LIN {X 0,Y 406.447,Z 396.018,A -85,B 0,C 180,E1 17983.42,E2 17983.42} C_VEL
LIN {X 0,Y 407.106,Z 396.844,A -85,B 0,C 180,E1 17981.451,E2 17981.451} C_VEL
LIN {X 0,Y 409.582,Z 400.807,A -85,B 0,C 180,E1 17978.37,E2 17978.37} C_VEL
LIN {X 0,Y 412.361,Z 402.697,A -85,B 0,C 180,E1 17976.455,E2 17976.455} C_VEL
LIN {X 0,Y 414.579,Z 406.468,A -85,B 0,C 180,E1 17975.036,E2 17975.036} C_VEL
LIN {X 0,Y 417.386,Z 409.126,A -85,B 0,C 180,E1 17973.649,E2 17973.649} C_VEL
LIN {X 0,Y 421.803,Z 415.235,A -85,B 0,C 180,E1 17971.701,E2 17971.701} C_VEL
LIN {X 0,Y 425.14,Z 419.754,A -85,B 0,C 180,E1 17970.443,E2 17970.443} C_VEL
LIN {X 0,Y 429.609,Z 426.182,A -85,B 0,C 180,E1 17968.891,E2 17968.891} C_VEL
LIN {X 0,Y 436.176,Z 435.925,A -85,B 0,C 180,E1 17966.897,E2 17966.897} C_VEL
LIN {X 0,Y 443.079,Z 446.923,A -85,B 0,C 180,E1 17965.028,E2 17965.028} C_VEL
LIN {X 0,Y 450.903,Z 460.1,A -85,B 0,C 180,E1 17963.124,E2 17963.124} C_VEL
LIN {X 0,Y 451.957,Z 462.413,A -85,B 0,C 180,E1 17962.867,E2 17962.867} C_VEL
LIN {X 0,Y 443.085,Z 650.195,A -85,B 0,C 180,E1 17959.257,E2 17959.257} C_VEL
LIN {X 0,Y 439.216,Z 737.669,A -85,B 0,C 180,E1 17957.582,E2 17957.582} C_VEL
LIN {X 0,Y 437.021,Z 761.221,A -85,B 0,C 180,E1 17956.942,E2 17956.942} C_VEL
LIN {X 0,Y 434.323,Z 783.972,A -85,B 0,C 180,E1 17956.104,E2 17956.104} C_VEL
LIN {X 0,Y 431.268,Z 805.02,A -85,B 0,C 180,E1 17955.098,E2 17955.098} C_VEL
LIN {X 0,Y 427.411,Z 828.313,A -85,B 0,C 180,E1 17953.71,E2 17953.71} C_VEL
LIN {X 0,Y 423.869,Z 847.343,A -85,B 0,C 180,E1 17952.338,E2 17952.338} C_VEL
LIN {X 0,Y 419.579,Z 868.496,A -85,B 0,C 180,E1 17950.521,E2 17950.521} C_VEL
LIN {X 0,Y 415.449,Z 887.81,A -85,B 0,C 180,E1 17948.563,E2 17948.563} C_VEL
LIN {X 0,Y 411.376,Z 906.017,A -85,B 0,C 180,E1 17946.377,E2 17946.377} C_VEL
LIN {X 0,Y 407.459,Z 923.411,A -85,B 0,C 180,E1 17943.962,E2 17943.962} C_VEL
LIN {X 0,Y 404.032,Z 938.688,A -85,B 0,C 180,E1 17941.481,E2 17941.481} C_VEL
LIN {X 0,Y 400.669,Z 954.261,A -85,B 0,C 180,E1 17938.55,E2 17938.55} C_VEL
LIN {X 0,Y 398.109,Z 966.963,A -85,B 0,C 180,E1 17935.756,E2 17935.756} C_VEL
LIN {X 0,Y 395.862,Z 979.241,A -85,B 0,C 180,E1 17932.58,E2 17932.58} C_VEL
LIN {X 0,Y 394.305,Z 989.174,A -85,B 0,C 180,E1 17929.559,E2 17929.559} C_VEL
LIN {X 0,Y 393.186,Z 997.73,A -85,B 0,C 180,E1 17926.399,E2 17926.399} C_VEL
LIN {X 0,Y 392.494,Z 1004.736,A -85,B 0,C 180,E1 17923.258,E2 17923.258} C_VEL
LIN {X 0,Y 392.088,Z 1010.3,A -85,B 0,C 180,E1 17919.989,E2 17919.989} C_VEL
LIN {X 0,Y 391.941,Z 1013.854,A -85,B 0,C 180,E1 17917.184,E2 17917.184} C_VEL
LIN {X 0,Y 391.914,Z 1016.518,A -85,B 0,C 180,E1 17913.954,E2 17913.954} C_VEL
LIN {X 0,Y 391.905,Z 1017.533,A -85,B 0,C 180,E1 17911.173,E2 17911.173} C_VEL
LIN {X 0,Y 391.911,Z 1017.466,A -85,B 0,C 180,E1 17908.396,E2 17908.396} C_VEL
LIN {X 0,Y 391.917,Z 1015.846,A -85,B 0,C 180,E1 17905.028,E2 17905.028} C_VEL
LIN {X 0,Y 391.978,Z 1013.228,A -85,B 0,C 180,E1 17902.234,E2 17902.234} C_VEL
LIN {X 0,Y 392.194,Z 1008.814,A -85,B 0,C 180,E1 17898.981,E2 17898.981} C_VEL
LIN {X 0,Y 392.64,Z 1002.949,A -85,B 0,C 180,E1 17895.854,E2 17895.854} C_VEL
LIN {X 0,Y 393.449,Z 995.665,A -85,B 0,C 180,E1 17892.707,E2 17892.707} C_VEL
LIN {X 0,Y 394.712,Z 986.541,A -85,B 0,C 180,E1 17889.544,E2 17889.544} C_VEL
LIN {X 0,Y 396.55,Z 975.718,A -85,B 0,C 180,E1 17886.37,E2 17886.37} C_VEL
LIN {X 0,Y 398.776,Z 964.082,A -85,B 0,C 180,E1 17883.498,E2 17883.498} C_VEL
LIN {X 0,Y 401.77,Z 949.865,A -85,B 0,C 180,E1 17880.484,E2 17880.484} C_VEL
LIN {X 0,Y 404.955,Z 935.505,A -85,B 0,C 180,E1 17877.874,E2 17877.874} C_VEL
LIN {X 0,Y 408.783,Z 918.746,A -85,B 0,C 180,E1 17875.262,E2 17875.262} C_VEL
LIN {X 0,Y 412.641,Z 901.934,A -85,B 0,C 180,E1 17872.999,E2 17872.999} C_VEL
LIN {X 0,Y 416.749,Z 883.443,A -85,B 0,C 180,E1 17870.883,E2 17870.883} C_VEL
LIN {X 0,Y 420.829,Z 864.613,A -85,B 0,C 180,E1 17869.03,E2 17869.03} C_VEL
LIN {X 0,Y 424.656,Z 845.158,A -85,B 0,C 180,E1 17867.422,E2 17867.422} C_VEL
LIN {X 0,Y 428.329,Z 825.276,A -85,B 0,C 180,E1 17866.023,E2 17866.023} C_VEL
LIN {X 0,Y 431.758,Z 803.746,A -85,B 0,C 180,E1 17864.789,E2 17864.789} C_VEL
LIN {X 0,Y 434.972,Z 780.771,A -85,B 0,C 180,E1 17863.734,E2 17863.734} C_VEL
LIN {X 0,Y 437.348,Z 759.57,A -85,B 0,C 180,E1 17862.988,E2 17862.988} C_VEL
LIN {X 0,Y 439.399,Z 734.535,A -85,B 0,C 180,E1 17862.352,E2 17862.352} C_VEL
LIN {X 0,Y 448.069,Z 525.057,A -85,B 0,C 180,E1 17858.43,E2 17858.43} C_VEL
LIN {X 0,Y 450.713,Z 461.917,A -85,B 0,C 180,E1 17857.213,E2 17857.213} C_VEL
LIN {X 0,Y 440.051,Z 445.277,A -85,B 0,C 180,E1 17854.969,E2 17854.969} C_VEL
LIN {X 0,Y 429.028,Z 429.211,A -85,B 0,C 180,E1 17852.452,E2 17852.452} C_VEL
LIN {X 0,Y 421.006,Z 418.219,A -85,B 0,C 180,E1 17850.467,E2 17850.467} C_VEL
LIN {X 0,Y 413.797,Z 408.572,A -85,B 0,C 180,E1 17848.543,E2 17848.543} C_VEL
LIN {X 0,Y 410.464,Z 404.237,A -85,B 0,C 180,E1 17847.608,E2 17847.608} C_VEL
LIN {X 0,Y 406.022,Z 398.588,A -85,B 0,C 180,E1 17846.312,E2 17846.312} C_VEL
LIN {X 0,Y 401.849,Z 393.423,A -85,B 0,C 180,E1 17845.023,E2 17845.023} C_VEL
LIN {X 0,Y 398.003,Z 388.428,A -85,B 0,C 180,E1 17843.778,E2 17843.778} C_VEL
LIN {X 0,Y 394.851,Z 385.59,A -85,B 0,C 180,E1 17842.755,E2 17842.755} C_VEL
LIN {X 0,Y 393.726,Z 383.145,A -85,B 0,C 180,E1 17842.233,E2 17842.233} C_VEL
LIN {X 0,Y 393.56,Z 382.126,A -85,B 0,C 180,E1 17841.772,E2 17841.772} C_VEL
LIN {X 0,Y 393.536,Z 382.017,A -85,B 0,C 180,E1 17837.7,E2 17837.7} C_VEL
LIN {X 0,Y 393.524,Z 382.017,A -85,B 0,C 180,E1 17833.817,E2 17833.817} C_VEL
LIN {X 0,Y 393.51,Z 382.027,A -85,B 0,C 180,E1 17829.949,E2 17829.949} C_VEL
LIN {X 0,Y 393.504,Z 382.032,A -85,B 0,C 180,E1 17826.126,E2 17826.126} C_VEL
LIN {X 0,Y 393.503,Z 382.025,A -85,B 0,C 180,E1 17822.184,E2 17822.184} C_VEL
LIN {X 0,Y 393.507,Z 382.019,A -85,B 0,C 180,E1 17818.252,E2 17818.252} C_VEL
LIN {X 0,Y 393.516,Z 382.015,A -85,B 0,C 180,E1 17814.313,E2 17814.313} C_VEL
LIN {X 0,Y 393.537,Z 382.014,A -85,B 0,C 180,E1 17810.494,E2 17810.494} C_VEL
LIN {X 0,Y 393.558,Z 382.012,A -85,B 0,C 180,E1 17806.632,E2 17806.632} C_VEL
LIN {X 0,Y 393.558,Z 382.015,A -85,B 0,C 180,E1 17802.707,E2 17802.707} C_VEL
LIN {X 0,Y 393.559,Z 382.02,A -85,B 0,C 180,E1 17798.697,E2 17798.697} C_VEL
LIN {X 0,Y 393.552,Z 382.026,A -85,B 0,C 180,E1 17794.734,E2 17794.734} C_VEL
LIN {X 0,Y 393.542,Z 382.027,A -85,B 0,C 180,E1 17790.803,E2 17790.803} C_VEL
LIN {X 0,Y 393.535,Z 382.021,A -85,B 0,C 180,E1 17786.889,E2 17786.889} C_VEL
LIN {X 0,Y 393.531,Z 382.016,A -85,B 0,C 180,E1 17782.911,E2 17782.911} C_VEL
LIN {X 0,Y 393.535,Z 382.014,A -85,B 0,C 180,E1 17778.981,E2 17778.981} C_VEL
LIN {X 0,Y 393.539,Z 382.025,A -85,B 0,C 180,E1 17774.928,E2 17774.928} C_VEL
LIN {X 0,Y 393.544,Z 382.021,A -85,B 0,C 180,E1 17770.95,E2 17770.95} C_VEL
LIN {X 0,Y 393.55,Z 382.014,A -85,B 0,C 180,E1 17767.016,E2 17767.016} C_VEL
LIN {X 0,Y 393.585,Z 382.191,A -85,B 0,C 180,E1 17765.366,E2 17765.366} C_VEL
LIN {X 0,Y 393.904,Z 383.571,A -85,B 0,C 180,E1 17764.927,E2 17764.927} C_VEL
LIN {X 0,Y 395.652,Z 386.503,A -85,B 0,C 180,E1 17764.272,E2 17764.272} C_VEL
LIN {X 0,Y 398.818,Z 388.946,A -85,B 0,C 180,E1 17763.281,E2 17763.281} C_VEL
LIN {X 0,Y 401.093,Z 392.587,A -85,B 0,C 180,E1 17762.52,E2 17762.52} C_VEL
LIN {X 0,Y 404.021,Z 395.14,A -85,B 0,C 180,E1 17761.639,E2 17761.639} C_VEL
LIN {X 0,Y 406.774,Z 399.093,A -85,B 0,C 180,E1 17760.786,E2 17760.786} C_VEL
LIN {X 0,Y 409.03,Z 401.334,A -85,B 0,C 180,E1 17760.148,E2 17760.148} C_VEL
LIN {X 0,Y 412.363,Z 405.67,A -85,B 0,C 180,E1 17759.203,E2 17759.203} C_VEL
LIN {X 0,Y 414.226,Z 407.789,A -85,B 0,C 180,E1 17758.703,E2 17758.703} C_VEL
LIN {X 0,Y 419.171,Z 413.919,A -85,B 0,C 180,E1 17757.406,E2 17757.406} C_VEL
LIN {X 0,Y 423.928,Z 420.03,A -85,B 0,C 180,E1 17756.204,E2 17756.204} C_VEL
LIN {X 0,Y 431.744,Z 430.135,A -85,B 0,C 180,E1 17754.34,E2 17754.34} C_VEL
LIN {X 0,Y 442.645,Z 445.003,A -85,B 0,C 180,E1 17751.946,E2 17751.946} C_VEL
LIN {X 0,Y 450.53,Z 456.58,A -85,B 0,C 180,E1 17750.328,E2 17750.328} C_VEL
LIN {X 0,Y 442.652,Z 641.056,A -85,B 0,C 180,E1 17746.873,E2 17746.873} C_VEL
LIN {X 0,Y 441.678,Z 648.751,A -85,B 0,C 180,E1 17746.826,E2 17746.826} C_VEL
LIN {X 0,Y 436.634,Z 669.324,A -85,B 0,C 180,E1 17747.051,E2 17747.051} C_VEL
LIN {X 0,Y 435.857,Z 675.927,A -85,B 0,C 180,E1 17747,E2 17747} C_VEL
LIN {X 0,Y 433.839,Z 717.756,A -85,B 0,C 180,E1 17746.18,E2 17746.18} C_VEL
LIN {X 0,Y 431.82,Z 739.993,A -85,B 0,C 180,E1 17745.546,E2 17745.546} C_VEL
LIN {X 0,Y 429.069,Z 763.419,A -85,B 0,C 180,E1 17744.641,E2 17744.641} C_VEL
LIN {X 0,Y 426.277,Z 782.547,A -85,B 0,C 180,E1 17743.7,E2 17743.7} C_VEL
LIN {X 0,Y 422.53,Z 804.668,A -85,B 0,C 180,E1 17742.362,E2 17742.362} C_VEL
LIN {X 0,Y 418.935,Z 823.202,A -85,B 0,C 180,E1 17741.003,E2 17741.003} C_VEL
LIN {X 0,Y 414.415,Z 844.319,A -85,B 0,C 180,E1 17739.159,E2 17739.159} C_VEL
LIN {X 0,Y 410.247,Z 862.498,A -85,B 0,C 180,E1 17737.274,E2 17737.274} C_VEL
LIN {X 0,Y 405.893,Z 880.407,A -85,B 0,C 180,E1 17735.084,E2 17735.084} C_VEL
LIN {X 0,Y 401.728,Z 897.125,A -85,B 0,C 180,E1 17732.707,E2 17732.707} C_VEL
LIN {X 0,Y 397.837,Z 912.385,A -85,B 0,C 180,E1 17730.14,E2 17730.14} C_VEL
LIN {X 0,Y 394.34,Z 926.605,A -85,B 0,C 180,E1 17727.38,E2 17727.38} C_VEL
LIN {X 0,Y 391.42,Z 938.864,A -85,B 0,C 180,E1 17724.573,E2 17724.573} C_VEL
LIN {X 0,Y 388.851,Z 950.67,A -85,B 0,C 180,E1 17721.42,E2 17721.42} C_VEL
LIN {X 0,Y 386.984,Z 960.23,A -85,B 0,C 180,E1 17718.37,E2 17718.37} C_VEL
LIN {X 0,Y 385.494,Z 969.457,A -85,B 0,C 180,E1 17714.81,E2 17714.81} C_VEL
LIN {X 0,Y 384.655,Z 976.186,A -85,B 0,C 180,E1 17711.582,E2 17711.582} C_VEL
LIN {X 0,Y 384.17,Z 981.649,A -85,B 0,C 180,E1 17708.147,E2 17708.147} C_VEL
LIN {X 0,Y 383.977,Z 985.556,A -85,B 0,C 180,E1 17704.716,E2 17704.716} C_VEL
LIN {X 0,Y 383.93,Z 987.8,A -85,B 0,C 180,E1 17701.36,E2 17701.36} C_VEL
LIN {X 0,Y 383.915,Z 988.609,A -85,B 0,C 180,E1 17698.08,E2 17698.08} C_VEL
LIN {X 0,Y 383.926,Z 987.87,A -85,B 0,C 180,E1 17694.676,E2 17694.676} C_VEL
LIN {X 0,Y 383.978,Z 985.703,A -85,B 0,C 180,E1 17691.318,E2 17691.318} C_VEL
LIN {X 0,Y 384.167,Z 981.866,A -85,B 0,C 180,E1 17687.882,E2 17687.882} C_VEL
LIN {X 0,Y 384.636,Z 976.512,A -85,B 0,C 180,E1 17684.451,E2 17684.451} C_VEL
LIN {X 0,Y 385.471,Z 969.833,A -85,B 0,C 180,E1 17681.212,E2 17681.212} C_VEL
LIN {X 0,Y 386.915,Z 960.986,A -85,B 0,C 180,E1 17677.74,E2 17677.74} C_VEL
LIN {X 0,Y 388.714,Z 951.69,A -85,B 0,C 180,E1 17674.735,E2 17674.735} C_VEL
LIN {X 0,Y 391.407,Z 939.423,A -85,B 0,C 180,E1 17671.408,E2 17671.408} C_VEL
LIN {X 0,Y 394.527,Z 926.457,A -85,B 0,C 180,E1 17668.425,E2 17668.425} C_VEL
LIN {X 0,Y 398.171,Z 911.785,A -85,B 0,C 180,E1 17665.59,E2 17665.59} C_VEL
LIN {X 0,Y 402.352,Z 895.45,A -85,B 0,C 180,E1 17662.886,E2 17662.886} C_VEL
LIN {X 0,Y 406.463,Z 879.226,A -85,B 0,C 180,E1 17660.596,E2 17660.596} C_VEL
LIN {X 0,Y 410.926,Z 860.86,A -85,B 0,C 180,E1 17658.383,E2 17658.383} C_VEL
LIN {X 0,Y 415.401,Z 841.777,A -85,B 0,C 180,E1 17656.429,E2 17656.429} C_VEL
LIN {X 0,Y 419.495,Z 822.459,A -85,B 0,C 180,E1 17654.776,E2 17654.776} C_VEL
LIN {X 0,Y 423.374,Z 802.677,A -85,B 0,C 180,E1 17653.339,E2 17653.339} C_VEL
LIN {X 0,Y 426.861,Z 781.831,A -85,B 0,C 180,E1 17652.102,E2 17652.102} C_VEL
LIN {X 0,Y 430.013,Z 760.158,A -85,B 0,C 180,E1 17651.053,E2 17651.053} C_VEL
LIN {X 0,Y 432.527,Z 738.038,A -85,B 0,C 180,E1 17650.233,E2 17650.233} C_VEL
LIN {X 0,Y 434.647,Z 712.891,A -85,B 0,C 180,E1 17649.563,E2 17649.563} C_VEL
LIN {X 0,Y 444.951,Z 502.944,A -85,B 0,C 180,E1 17645.5,E2 17645.5} C_VEL
LIN {X 0,Y 447.109,Z 460.805,A -85,B 0,C 180,E1 17644.65,E2 17644.65} C_VEL
LIN {X 0,Y 439.45,Z 449.084,A -85,B 0,C 180,E1 17642.739,E2 17642.739} C_VEL
LIN {X 0,Y 432.726,Z 439.435,A -85,B 0,C 180,E1 17640.861,E2 17640.861} C_VEL
LIN {X 0,Y 426.889,Z 431.418,A -85,B 0,C 180,E1 17639.027,E2 17639.027} C_VEL
LIN {X 0,Y 423.277,Z 426.612,A -85,B 0,C 180,E1 17637.75,E2 17637.75} C_VEL
LIN {X 0,Y 419.427,Z 421.563,A -85,B 0,C 180,E1 17636.242,E2 17636.242} C_VEL
LIN {X 0,Y 416.196,Z 417.577,A -85,B 0,C 180,E1 17634.797,E2 17634.797} C_VEL
LIN {X 0,Y 415.277,Z 416.109,A -85,B 0,C 180,E1 17634.335,E2 17634.335} C_VEL
LIN {X 0,Y 412.079,Z 412.864,A -85,B 0,C 180,E1 17632.612,E2 17632.612} C_VEL
LIN {X 0,Y 410.451,Z 410.075,A -85,B 0,C 180,E1 17631.511,E2 17631.511} C_VEL
LIN {X 0,Y 406.913,Z 407.011,A -85,B 0,C 180,E1 17628.52,E2 17628.52} C_VEL
LIN {X 0,Y 405.709,Z 404.273,A -85,B 0,C 180,E1 17626.315,E2 17626.315} C_VEL
LIN {X 0,Y 405.34,Z 403.948,A -85,B 0,C 180,E1 17623.374,E2 17623.374} C_VEL
LIN {X 0,Y 405.911,Z 404.661,A -85,B 0,C 180,E1 17621.622,E2 17621.622} C_VEL
LIN {X 0,Y 408.352,Z 408.698,A -85,B 0,C 180,E1 17618.453,E2 17618.453} C_VEL
LIN {X 0,Y 410.84,Z 410.578,A -85,B 0,C 180,E1 17616.667,E2 17616.667} C_VEL
LIN {X 0,Y 413.282,Z 414.449,A -85,B 0,C 180,E1 17615.105,E2 17615.105} C_VEL
LIN {X 0,Y 415.69,Z 416.816,A -85,B 0,C 180,E1 17613.886,E2 17613.886} C_VEL
LIN {X 0,Y 419.948,Z 422.878,A -85,B 0,C 180,E1 17611.951,E2 17611.951} C_VEL
LIN {X 0,Y 422.937,Z 427.073,A -85,B 0,C 180,E1 17610.779,E2 17610.779} C_VEL
LIN {X 0,Y 428.371,Z 434.95,A -85,B 0,C 180,E1 17608.869,E2 17608.869} C_VEL
LIN {X 0,Y 435.097,Z 445.542,A -85,B 0,C 180,E1 17606.805,E2 17606.805} C_VEL
LIN {X 0,Y 441.885,Z 456.681,A -85,B 0,C 180,E1 17604.96,E2 17604.96} C_VEL
LIN {X 0,Y 447.17,Z 466.131,A -85,B 0,C 180,E1 17603.635,E2 17603.635} C_VEL
LIN {X 0,Y 437.799,Z 653.274,A -85,B 0,C 180,E1 17600,E2 17600} C_VEL
LIN {X 0,Y 433.839,Z 737.361,A -85,B 0,C 180,E1 17598.368,E2 17598.368} C_VEL
LIN {X 0,Y 431.556,Z 760.907,A -85,B 0,C 180,E1 17597.724,E2 17597.724} C_VEL
LIN {X 0,Y 428.741,Z 783.618,A -85,B 0,C 180,E1 17596.884,E2 17596.884} C_VEL
LIN {X 0,Y 425.543,Z 804.601,A -85,B 0,C 180,E1 17595.876,E2 17595.876} C_VEL
LIN {X 0,Y 421.46,Z 828.087,A -85,B 0,C 180,E1 17594.468,E2 17594.468} C_VEL
LIN {X 0,Y 417.618,Z 847.811,A -85,B 0,C 180,E1 17593.03,E2 17593.03} C_VEL
LIN {X 0,Y 413.324,Z 867.93,A -85,B 0,C 180,E1 17591.278,E2 17591.278} C_VEL
LIN {X 0,Y 409.099,Z 886.671,A -85,B 0,C 180,E1 17589.366,E2 17589.366} C_VEL
LIN {X 0,Y 404.842,Z 904.725,A -85,B 0,C 180,E1 17587.19,E2 17587.19} C_VEL
LIN {X 0,Y 400.727,Z 922.148,A -85,B 0,C 180,E1 17584.763,E2 17584.763} C_VEL
LIN {X 0,Y 396.867,Z 938.245,A -85,B 0,C 180,E1 17582.116,E2 17582.116} C_VEL
LIN {X 0,Y 393.38,Z 953.475,A -85,B 0,C 180,E1 17579.213,E2 17579.213} C_VEL
LIN {X 0,Y 390.649,Z 966.145,A -85,B 0,C 180,E1 17576.388,E2 17576.388} C_VEL
LIN {X 0,Y 388.161,Z 978.857,A -85,B 0,C 180,E1 17573.053,E2 17573.053} C_VEL
LIN {X 0,Y 386.486,Z 988.803,A -85,B 0,C 180,E1 17569.971,E2 17569.971} C_VEL
LIN {X 0,Y 385.282,Z 997.376,A -85,B 0,C 180,E1 17566.745,E2 17566.745} C_VEL
LIN {X 0,Y 384.563,Z 1004.083,A -85,B 0,C 180,E1 17563.689,E2 17563.689} C_VEL
LIN {X 0,Y 384.114,Z 1009.854,A -85,B 0,C 180,E1 17560.284,E2 17560.284} C_VEL
LIN {X 0,Y 383.956,Z 1013.372,A -85,B 0,C 180,E1 17557.485,E2 17557.485} C_VEL
LIN {X 0,Y 383.917,Z 1016.07,A -85,B 0,C 180,E1 17554.335,E2 17554.335} C_VEL
LIN {X 0,Y 383.916,Z 1017.207,A -85,B 0,C 180,E1 17551.347,E2 17551.347} C_VEL
LIN {X 0,Y 383.917,Z 1017.19,A -85,B 0,C 180,E1 17548.512,E2 17548.512} C_VEL
LIN {X 0,Y 383.917,Z 1015.781,A -85,B 0,C 180,E1 17545.224,E2 17545.224} C_VEL
LIN {X 0,Y 383.979,Z 1013.093,A -85,B 0,C 180,E1 17542.222,E2 17542.222} C_VEL
LIN {X 0,Y 384.187,Z 1008.986,A -85,B 0,C 180,E1 17539.052,E2 17539.052} C_VEL
LIN {X 0,Y 384.645,Z 1003.203,A -85,B 0,C 180,E1 17535.831,E2 17535.831} C_VEL
LIN {X 0,Y 385.421,Z 996.454,A -85,B 0,C 180,E1 17532.803,E2 17532.803} C_VEL
LIN {X 0,Y 386.78,Z 987.158,A -85,B 0,C 180,E1 17529.421,E2 17529.421} C_VEL
LIN {X 0,Y 388.585,Z 977.068,A -85,B 0,C 180,E1 17526.339,E2 17526.339} C_VEL
LIN {X 0,Y 391.007,Z 965.039,A -85,B 0,C 180,E1 17523.258,E2 17523.258} C_VEL
LIN {X 0,Y 393.96,Z 951.86,A -85,B 0,C 180,E1 17520.342,E2 17520.342} C_VEL
LIN {X 0,Y 397.35,Z 937.204,A -85,B 0,C 180,E1 17517.596,E2 17517.596} C_VEL
LIN {X 0,Y 401.426,Z 920.406,A -85,B 0,C 180,E1 17514.881,E2 17514.881} C_VEL
LIN {X 0,Y 405.309,Z 904.242,A -85,B 0,C 180,E1 17512.644,E2 17512.644} C_VEL
LIN {X 0,Y 409.892,Z 884.772,A -85,B 0,C 180,E1 17510.343,E2 17510.343} C_VEL
LIN {X 0,Y 414.085,Z 866.277,A -85,B 0,C 180,E1 17508.483,E2 17508.483} C_VEL
LIN {X 0,Y 418.252,Z 846.309,A -85,B 0,C 180,E1 17506.789,E2 17506.789} C_VEL
LIN {X 0,Y 422.24,Z 825.708,A -85,B 0,C 180,E1 17505.315,E2 17505.315} C_VEL
LIN {X 0,Y 425.93,Z 803.593,A -85,B 0,C 180,E1 17504.037,E2 17504.037} C_VEL
LIN {X 0,Y 429.289,Z 780.498,A -85,B 0,C 180,E1 17502.972,E2 17502.972} C_VEL
LIN {X 0,Y 431.714,Z 759.649,A -85,B 0,C 180,E1 17502.236,E2 17502.236} C_VEL
LIN {X 0,Y 433.861,Z 734.539,A -85,B 0,C 180,E1 17501.59,E2 17501.59} C_VEL
LIN {X 0,Y 442.99,Z 525.076,A -85,B 0,C 180,E1 17497.63,E2 17497.63} C_VEL
LIN {X 0,Y 445.609,Z 465.785,A -85,B 0,C 180,E1 17496.484,E2 17496.484} C_VEL
LIN {X 0,Y 434.795,Z 448.963,A -85,B 0,C 180,E1 17494.132,E2 17494.132} C_VEL
LIN {X 0,Y 424.828,Z 434.413,A -85,B 0,C 180,E1 17491.776,E2 17491.776} C_VEL
LIN {X 0,Y 415.337,Z 421.227,A -85,B 0,C 180,E1 17489.333,E2 17489.333} C_VEL
LIN {X 0,Y 407.646,Z 411.108,A -85,B 0,C 180,E1 17487.182,E2 17487.182} C_VEL
LIN {X 0,Y 403.271,Z 405.482,A -85,B 0,C 180,E1 17485.872,E2 17485.872} C_VEL
LIN {X 0,Y 399.227,Z 400.458,A -85,B 0,C 180,E1 17484.605,E2 17484.605} C_VEL
LIN {X 0,Y 395.116,Z 395.318,A -85,B 0,C 180,E1 17483.251,E2 17483.251} C_VEL
LIN {X 0,Y 392.162,Z 392.283,A -85,B 0,C 180,E1 17482.247,E2 17482.247} C_VEL
LIN {X 0,Y 390.555,Z 389.517,A -85,B 0,C 180,E1 17481.632,E2 17481.632} C_VEL
LIN {X 0,Y 387.32,Z 387.115,A -85,B 0,C 180,E1 17480.513,E2 17480.513} C_VEL
LIN {X 0,Y 385.698,Z 383.627,A -85,B 0,C 180,E1 17479.694,E2 17479.694} C_VEL
LIN {X 0,Y 385.566,Z 383.038,A -85,B 0,C 180,E1 17479.071,E2 17479.071} C_VEL
LIN {X 0,Y 385.577,Z 383.013,A -85,B 0,C 180,E1 17475.183,E2 17475.183} C_VEL
LIN {X 0,Y 385.59,Z 383.004,A -85,B 0,C 180,E1 17471.214,E2 17471.214} C_VEL
LIN {X 0,Y 385.602,Z 383.005,A -85,B 0,C 180,E1 17467.149,E2 17467.149} C_VEL
LIN {X 0,Y 385.604,Z 383.015,A -85,B 0,C 180,E1 17463.121,E2 17463.121} C_VEL
LIN {X 0,Y 385.619,Z 383.012,A -85,B 0,C 180,E1 17459.108,E2 17459.108} C_VEL
LIN {X 0,Y 385.613,Z 383.003,A -85,B 0,C 180,E1 17454.942,E2 17454.942} C_VEL
LIN {X 0,Y 385.616,Z 383,A -85,B 0,C 180,E1 17450.899,E2 17450.899} C_VEL
LIN {X 0,Y 385.619,Z 383,A -85,B 0,C 180,E1 17446.81,E2 17446.81} C_VEL
LIN {X 0,Y 385.615,Z 383.002,A -85,B 0,C 180,E1 17442.807,E2 17442.807} C_VEL
LIN {X 0,Y 385.619,Z 383.008,A -85,B 0,C 180,E1 17438.715,E2 17438.715} C_VEL
LIN {X 0,Y 385.616,Z 383.016,A -85,B 0,C 180,E1 17434.67,E2 17434.67} C_VEL
LIN {X 0,Y 385.618,Z 383.01,A -85,B 0,C 180,E1 17430.587,E2 17430.587} C_VEL
LIN {X 0,Y 385.609,Z 383.004,A -85,B 0,C 180,E1 17426.598,E2 17426.598} C_VEL
LIN {X 0,Y 385.601,Z 383.003,A -85,B 0,C 180,E1 17422.644,E2 17422.644} C_VEL
LIN {X 0,Y 385.598,Z 383.004,A -85,B 0,C 180,E1 17418.753,E2 17418.753} C_VEL
LIN {X 0,Y 385.6,Z 383.017,A -85,B 0,C 180,E1 17414.725,E2 17414.725} C_VEL
LIN {X 0,Y 385.602,Z 383.008,A -85,B 0,C 180,E1 17410.786,E2 17410.786} C_VEL
LIN {X 0,Y 385.653,Z 383.205,A -85,B 0,C 180,E1 17407.835,E2 17407.835} C_VEL
LIN {X 0,Y 386.014,Z 384.671,A -85,B 0,C 180,E1 17407.326,E2 17407.326} C_VEL
LIN {X 0,Y 387.873,Z 387.663,A -85,B 0,C 180,E1 17406.571,E2 17406.571} C_VEL
LIN {X 0,Y 391.037,Z 389.979,A -85,B 0,C 180,E1 17405.492,E2 17405.492} C_VEL
LIN {X 0,Y 393.23,Z 393.627,A -85,B 0,C 180,E1 17404.67,E2 17404.67} C_VEL
LIN {X 0,Y 396.311,Z 396.274,A -85,B 0,C 180,E1 17403.672,E2 17403.672} C_VEL
LIN {X 0,Y 399.072,Z 400.199,A -85,B 0,C 180,E1 17402.758,E2 17402.758} C_VEL
LIN {X 0,Y 401.614,Z 402.613,A -85,B 0,C 180,E1 17401.983,E2 17401.983} C_VEL
LIN {X 0,Y 404.908,Z 406.874,A -85,B 0,C 180,E1 17400.964,E2 17400.964} C_VEL
LIN {X 0,Y 406.537,Z 408.711,A -85,B 0,C 180,E1 17400.488,E2 17400.488} C_VEL
LIN {X 0,Y 410.325,Z 413.324,A -85,B 0,C 180,E1 17399.408,E2 17399.408} C_VEL
LIN {X 0,Y 416.832,Z 421.557,A -85,B 0,C 180,E1 17397.659,E2 17397.659} C_VEL
LIN {X 0,Y 424.221,Z 431.022,A -85,B 0,C 180,E1 17395.796,E2 17395.796} C_VEL
LIN {X 0,Y 434.881,Z 445.379,A -85,B 0,C 180,E1 17393.311,E2 17393.311} C_VEL
LIN {X 0,Y 445.39,Z 460.469,A -85,B 0,C 180,E1 17391.063,E2 17391.063} C_VEL
LIN {X 0,Y 436.207,Z 667.494,A -85,B 0,C 180,E1 17387.158,E2 17387.158} C_VEL
LIN {X 0,Y 435.857,Z 675.927,A -85,B 0,C 180,E1 17387,E2 17387} C_VEL
LIN {X 0,Y 434.871,Z 683.623,A -85,B 0,C 180,E1 17386.953,E2 17386.953} C_VEL
LIN {X 0,Y 429.736,Z 704.174,A -85,B 0,C 180,E1 17387.186,E2 17387.186} C_VEL
LIN {X 0,Y 428.865,Z 710.76,A -85,B 0,C 180,E1 17387.118,E2 17387.118} C_VEL
LIN {X 0,Y 426.871,Z 734.858,A -85,B 0,C 180,E1 17386.499,E2 17386.499} C_VEL
LIN {X 0,Y 424.362,Z 756.652,A -85,B 0,C 180,E1 17385.717,E2 17385.717} C_VEL
LIN {X 0,Y 421.06,Z 779.51,A -85,B 0,C 180,E1 17384.645,E2 17384.645} C_VEL
LIN {X 0,Y 417.521,Z 800.347,A -85,B 0,C 180,E1 17383.428,E2 17383.428} C_VEL
LIN {X 0,Y 413.555,Z 820.382,A -85,B 0,C 180,E1 17381.997,E2 17381.997} C_VEL
LIN {X 0,Y 409.354,Z 839.853,A -85,B 0,C 180,E1 17380.348,E2 17380.348} C_VEL
LIN {X 0,Y 404.839,Z 858.634,A -85,B 0,C 180,E1 17378.446,E2 17378.446} C_VEL
LIN {X 0,Y 400.319,Z 876.744,A -85,B 0,C 180,E1 17376.305,E2 17376.305} C_VEL
LIN {X 0,Y 396.074,Z 892.878,A -85,B 0,C 180,E1 17374.049,E2 17374.049} C_VEL
LIN {X 0,Y 391.833,Z 908.891,A -85,B 0,C 180,E1 17371.458,E2 17371.458} C_VEL
LIN {X 0,Y 388.044,Z 923.21,A -85,B 0,C 180,E1 17368.726,E2 17368.726} C_VEL
LIN {X 0,Y 384.406,Z 937.503,A -85,B 0,C 180,E1 17365.521,E2 17365.521} C_VEL
LIN {X 0,Y 381.697,Z 949.045,A -85,B 0,C 180,E1 17362.47,E2 17362.47} C_VEL
LIN {X 0,Y 379.499,Z 959.302,A -85,B 0,C 180,E1 17359.215,E2 17359.215} C_VEL
LIN {X 0,Y 377.942,Z 968.074,A -85,B 0,C 180,E1 17355.91,E2 17355.91} C_VEL
LIN {X 0,Y 376.903,Z 975.155,A -85,B 0,C 180,E1 17352.553,E2 17352.553} C_VEL
LIN {X 0,Y 376.301,Z 980.907,A -85,B 0,C 180,E1 17349.139,E2 17349.139} C_VEL
LIN {X 0,Y 376.032,Z 984.932,A -85,B 0,C 180,E1 17345.788,E2 17345.788} C_VEL
LIN {X 0,Y 375.922,Z 987.626,A -85,B 0,C 180,E1 17342.429,E2 17342.429} C_VEL
LIN {X 0,Y 375.928,Z 988.764,A -85,B 0,C 180,E1 17339.111,E2 17339.111} C_VEL
LIN {X 0,Y 375.907,Z 988.635,A -85,B 0,C 180,E1 17335.814,E2 17335.814} C_VEL
LIN {X 0,Y 375.943,Z 986.94,A -85,B 0,C 180,E1 17332.426,E2 17332.426} C_VEL
LIN {X 0,Y 376.06,Z 984.129,A -85,B 0,C 180,E1 17329.267,E2 17329.267} C_VEL
LIN {X 0,Y 376.434,Z 979.521,A -85,B 0,C 180,E1 17325.821,E2 17325.821} C_VEL
LIN {X 0,Y 377.126,Z 973.693,A -85,B 0,C 180,E1 17322.516,E2 17322.516} C_VEL
LIN {X 0,Y 378.281,Z 966.178,A -85,B 0,C 180,E1 17319.177,E2 17319.177} C_VEL
LIN {X 0,Y 380.029,Z 957.15,A -85,B 0,C 180,E1 17315.866,E2 17315.866} C_VEL
LIN {X 0,Y 382.425,Z 946.257,A -85,B 0,C 180,E1 17312.588,E2 17312.588} C_VEL
LIN {X 0,Y 385.367,Z 934.359,A -85,B 0,C 180,E1 17309.536,E2 17309.536} C_VEL
LIN {X 0,Y 388.83,Z 920.939,A -85,B 0,C 180,E1 17306.634,E2 17306.634} C_VEL
LIN {X 0,Y 393.133,Z 904.961,A -85,B 0,C 180,E1 17303.694,E2 17303.694} C_VEL
LIN {X 0,Y 397.327,Z 889.407,A -85,B 0,C 180,E1 17301.246,E2 17301.246} C_VEL
LIN {X 0,Y 401.788,Z 872.41,A -85,B 0,C 180,E1 17298.973,E2 17298.973} C_VEL
LIN {X 0,Y 406.457,Z 854.139,A -85,B 0,C 180,E1 17296.874,E2 17296.874} C_VEL
LIN {X 0,Y 410.974,Z 834.728,A -85,B 0,C 180,E1 17295.008,E2 17295.008} C_VEL
LIN {X 0,Y 415.36,Z 814.48,A -85,B 0,C 180,E1 17293.362,E2 17293.362} C_VEL
LIN {X 0,Y 419.154,Z 794.607,A -85,B 0,C 180,E1 17292.027,E2 17292.027} C_VEL
LIN {X 0,Y 422.999,Z 771.437,A -85,B 0,C 180,E1 17290.763,E2 17290.763} C_VEL
LIN {X 0,Y 425.802,Z 751.103,A -85,B 0,C 180,E1 17289.883,E2 17289.883} C_VEL
LIN {X 0,Y 428.277,Z 727.942,A -85,B 0,C 180,E1 17289.124,E2 17289.124} C_VEL
LIN {X 0,Y 429.913,Z 705.731,A -85,B 0,C 180,E1 17288.599,E2 17288.599} C_VEL
LIN {X 0,Y 439.97,Z 510.245,A -85,B 0,C 180,E1 17284.789,E2 17284.789} C_VEL
LIN {X 0,Y 442.501,Z 465.076,A -85,B 0,C 180,E1 17283.887,E2 17283.887} C_VEL
LIN {X 0,Y 434.327,Z 452.505,A -85,B 0,C 180,E1 17281.715,E2 17281.715} C_VEL
LIN {X 0,Y 427.43,Z 442.632,A -85,B 0,C 180,E1 17279.632,E2 17279.632} C_VEL
LIN {X 0,Y 423.723,Z 437.533,A -85,B 0,C 180,E1 17278.378,E2 17278.378} C_VEL
LIN {X 0,Y 420.931,Z 433.714,A -85,B 0,C 180,E1 17277.346,E2 17277.346} C_VEL
LIN {X 0,Y 417.347,Z 428.895,A -85,B 0,C 180,E1 17275.879,E2 17275.879} C_VEL
LIN {X 0,Y 414.089,Z 424.604,A -85,B 0,C 180,E1 17274.354,E2 17274.354} C_VEL
LIN {X 0,Y 413.17,Z 423.466,A -85,B 0,C 180,E1 17273.888,E2 17273.888} C_VEL
LIN {X 0,Y 410.071,Z 419.827,A -85,B 0,C 180,E1 17272.082,E2 17272.082} C_VEL
LIN {X 0,Y 408.955,Z 417.84,A -85,B 0,C 180,E1 17271.282,E2 17271.282} C_VEL
LIN {X 0,Y 405.642,Z 414.805,A -85,B 0,C 180,E1 17268.34,E2 17268.34} C_VEL
LIN {X 0,Y 404.561,Z 412.177,A -85,B 0,C 180,E1 17266.243,E2 17266.243} C_VEL
LIN {X 0,Y 404.233,Z 411.878,A -85,B 0,C 180,E1 17263.327,E2 17263.327} C_VEL
LIN {X 0,Y 404.748,Z 412.566,A -85,B 0,C 180,E1 17261.716,E2 17261.716} C_VEL
LIN {X 0,Y 406.96,Z 416.441,A -85,B 0,C 180,E1 17258.678,E2 17258.678} C_VEL
LIN {X 0,Y 409.284,Z 418.308,A -85,B 0,C 180,E1 17256.916,E2 17256.916} C_VEL
LIN {X 0,Y 411.988,Z 422.415,A -85,B 0,C 180,E1 17255.175,E2 17255.175} C_VEL
LIN {X 0,Y 413.946,Z 424.429,A -85,B 0,C 180,E1 17254.153,E2 17254.153} C_VEL
LIN {X 0,Y 418.18,Z 430.624,A -85,B 0,C 180,E1 17252.171,E2 17252.171} C_VEL
LIN {X 0,Y 420.929,Z 434.652,A -85,B 0,C 180,E1 17251.055,E2 17251.055} C_VEL
LIN {X 0,Y 425.891,Z 442.029,A -85,B 0,C 180,E1 17249.256,E2 17249.256} C_VEL
LIN {X 0,Y 432.353,Z 452.471,A -85,B 0,C 180,E1 17247.199,E2 17247.199} C_VEL
LIN {X 0,Y 438.764,Z 463.293,A -85,B 0,C 180,E1 17245.39,E2 17245.39} C_VEL
LIN {X 0,Y 442.477,Z 470.125,A -85,B 0,C 180,E1 17244.417,E2 17244.417} C_VEL
LIN {X 0,Y 432.675,Z 654.988,A -85,B 0,C 180,E1 17240.789,E2 17240.789} C_VEL
LIN {X 0,Y 428.561,Z 737.343,A -85,B 0,C 180,E1 17239.172,E2 17239.172} C_VEL
LIN {X 0,Y 426.183,Z 760.747,A -85,B 0,C 180,E1 17238.524,E2 17238.524} C_VEL
LIN {X 0,Y 423.222,Z 783.476,A -85,B 0,C 180,E1 17237.678,E2 17237.678} C_VEL
LIN {X 0,Y 419.697,Z 805.542,A -85,B 0,C 180,E1 17236.606,E2 17236.606} C_VEL
LIN {X 0,Y 415.531,Z 828.243,A -85,B 0,C 180,E1 17235.224,E2 17235.224} C_VEL
LIN {X 0,Y 411.433,Z 848.298,A -85,B 0,C 180,E1 17233.743,E2 17233.743} C_VEL
LIN {X 0,Y 406.878,Z 868.557,A -85,B 0,C 180,E1 17231.948,E2 17231.948} C_VEL
LIN {X 0,Y 402.372,Z 887.587,A -85,B 0,C 180,E1 17229.97,E2 17229.97} C_VEL
LIN {X 0,Y 397.846,Z 905.69,A -85,B 0,C 180,E1 17227.734,E2 17227.734} C_VEL
LIN {X 0,Y 393.471,Z 923.143,A -85,B 0,C 180,E1 17225.231,E2 17225.231} C_VEL
LIN {X 0,Y 389.549,Z 938.689,A -85,B 0,C 180,E1 17222.619,E2 17222.619} C_VEL
LIN {X 0,Y 385.709,Z 954.504,A -85,B 0,C 180,E1 17219.51,E2 17219.51} C_VEL
LIN {X 0,Y 382.789,Z 967.461,A -85,B 0,C 180,E1 17216.533,E2 17216.533} C_VEL
LIN {X 0,Y 380.378,Z 979.005,A -85,B 0,C 180,E1 17213.389,E2 17213.389} C_VEL
LIN {X 0,Y 378.542,Z 989.36,A -85,B 0,C 180,E1 17210.086,E2 17210.086} C_VEL
LIN {X 0,Y 377.296,Z 997.759,A -85,B 0,C 180,E1 17206.793,E2 17206.793} C_VEL
LIN {X 0,Y 376.535,Z 1004.669,A -85,B 0,C 180,E1 17203.517,E2 17203.517} C_VEL
LIN {X 0,Y 376.111,Z 1009.863,A -85,B 0,C 180,E1 17200.264,E2 17200.264} C_VEL
LIN {X 0,Y 375.95,Z 1013.39,A -85,B 0,C 180,E1 17197.338,E2 17197.338} C_VEL
LIN {X 0,Y 375.922,Z 1015.975,A -85,B 0,C 180,E1 17193.969,E2 17193.969} C_VEL
LIN {X 0,Y 375.911,Z 1016.951,A -85,B 0,C 180,E1 17191.071,E2 17191.071} C_VEL
LIN {X 0,Y 375.923,Z 1016.823,A -85,B 0,C 180,E1 17188.023,E2 17188.023} C_VEL
LIN {X 0,Y 375.927,Z 1015.132,A -85,B 0,C 180,E1 17184.663,E2 17184.663} C_VEL
LIN {X 0,Y 376.024,Z 1012.255,A -85,B 0,C 180,E1 17181.552,E2 17181.552} C_VEL
LIN {X 0,Y 376.291,Z 1007.422,A -85,B 0,C 180,E1 17178.043,E2 17178.043} C_VEL
LIN {X 0,Y 376.826,Z 1001.793,A -85,B 0,C 180,E1 17174.976,E2 17174.976} C_VEL
LIN {X 0,Y 377.895,Z 993.788,A -85,B 0,C 180,E1 17171.493,E2 17171.493} C_VEL
LIN {X 0,Y 379.363,Z 984.953,A -85,B 0,C 180,E1 17168.352,E2 17168.352} C_VEL
LIN {X 0,Y 381.663,Z 973.288,A -85,B 0,C 180,E1 17164.893,E2 17164.893} C_VEL
LIN {X 0,Y 384.472,Z 960.788,A -85,B 0,C 180,E1 17161.756,E2 17161.756} C_VEL
LIN {X 0,Y 387.791,Z 946.764,A -85,B 0,C 180,E1 17158.791,E2 17158.791} C_VEL
LIN {X 0,Y 391.766,Z 931.071,A -85,B 0,C 180,E1 17155.936,E2 17155.936} C_VEL
LIN {X 0,Y 395.616,Z 915.844,A -85,B 0,C 180,E1 17153.57,E2 17153.57} C_VEL
LIN {X 0,Y 400.304,Z 897.349,A -85,B 0,C 180,E1 17151.101,E2 17151.101} C_VEL
LIN {X 0,Y 404.493,Z 880.191,A -85,B 0,C 180,E1 17149.147,E2 17149.147} C_VEL
LIN {X 0,Y 409.31,Z 859.268,A -85,B 0,C 180,E1 17147.124,E2 17147.124} C_VEL
LIN {X 0,Y 413.698,Z 838.911,A -85,B 0,C 180,E1 17145.477,E2 17145.477} C_VEL
LIN {X 0,Y 417.644,Z 818.166,A -85,B 0,C 180,E1 17144.1,E2 17144.1} C_VEL
LIN {X 0,Y 421.368,Z 796.29,A -85,B 0,C 180,E1 17142.903,E2 17142.903} C_VEL
LIN {X 0,Y 424.379,Z 774.725,A -85,B 0,C 180,E1 17141.979,E2 17141.979} C_VEL
LIN {X 0,Y 426.96,Z 752.36,A -85,B 0,C 180,E1 17141.243,E2 17141.243} C_VEL
LIN {X 0,Y 428.699,Z 729.526,A -85,B 0,C 180,E1 17140.704,E2 17140.704} C_VEL
LIN {X 0,Y 438.232,Z 519.347,A -85,B 0,C 180,E1 17136.708,E2 17136.708} C_VEL
LIN {X 0,Y 440.498,Z 469.698,A -85,B 0,C 180,E1 17135.73,E2 17135.73} C_VEL
LIN {X 0,Y 430.593,Z 454.213,A -85,B 0,C 180,E1 17133.508,E2 17133.508} C_VEL
LIN {X 0,Y 419.842,Z 438.296,A -85,B 0,C 180,E1 17130.878,E2 17130.878} C_VEL
LIN {X 0,Y 408.673,Z 422.952,A -85,B 0,C 180,E1 17127.859,E2 17127.859} C_VEL
LIN {X 0,Y 404.094,Z 417.077,A -85,B 0,C 180,E1 17126.526,E2 17126.526} C_VEL
LIN {X 0,Y 400.535,Z 412.356,A -85,B 0,C 180,E1 17125.427,E2 17125.427} C_VEL
LIN {X 0,Y 396.311,Z 407.142,A -85,B 0,C 180,E1 17124.084,E2 17124.084} C_VEL
LIN {X 0,Y 392.667,Z 402.534,A -85,B 0,C 180,E1 17122.849,E2 17122.849} C_VEL
LIN {X 0,Y 389.58,Z 399.112,A -85,B 0,C 180,E1 17121.768,E2 17121.768} C_VEL
LIN {X 0,Y 388.121,Z 396.872,A -85,B 0,C 180,E1 17121.219,E2 17121.219} C_VEL
LIN {X 0,Y 384.974,Z 394.212,A -85,B 0,C 180,E1 17120.089,E2 17120.089} C_VEL
LIN {X 0,Y 382.894,Z 390.594,A -85,B 0,C 180,E1 17119.209,E2 17119.209} C_VEL
LIN {X 0,Y 379.774,Z 388.519,A -85,B 0,C 180,E1 17118.02,E2 17118.02} C_VEL
LIN {X 0,Y 377.844,Z 385.098,A -85,B 0,C 180,E1 17117.081,E2 17117.081} C_VEL
LIN {X 0,Y 377.622,Z 384.05,A -85,B 0,C 180,E1 17116.457,E2 17116.457} C_VEL
LIN {X 0,Y 377.619,Z 384.008,A -85,B 0,C 180,E1 17112.384,E2 17112.384} C_VEL
LIN {X 0,Y 377.62,Z 383.997,A -85,B 0,C 180,E1 17108.373,E2 17108.373} C_VEL
LIN {X 0,Y 377.624,Z 383.995,A -85,B 0,C 180,E1 17104.251,E2 17104.251} C_VEL
LIN {X 0,Y 377.629,Z 384.002,A -85,B 0,C 180,E1 17100.151,E2 17100.151} C_VEL
LIN {X 0,Y 377.633,Z 384.009,A -85,B 0,C 180,E1 17096.052,E2 17096.052} C_VEL
LIN {X 0,Y 377.636,Z 384.005,A -85,B 0,C 180,E1 17091.933,E2 17091.933} C_VEL
LIN {X 0,Y 377.638,Z 383.996,A -85,B 0,C 180,E1 17087.771,E2 17087.771} C_VEL
LIN {X 0,Y 377.64,Z 383.992,A -85,B 0,C 180,E1 17083.7,E2 17083.7} C_VEL
LIN {X 0,Y 377.644,Z 383.992,A -85,B 0,C 180,E1 17079.579,E2 17079.579} C_VEL
LIN {X 0,Y 377.648,Z 383.995,A -85,B 0,C 180,E1 17075.598,E2 17075.598} C_VEL
LIN {X 0,Y 377.653,Z 384.003,A -85,B 0,C 180,E1 17071.509,E2 17071.509} C_VEL
LIN {X 0,Y 377.659,Z 384.006,A -85,B 0,C 180,E1 17067.49,E2 17067.49} C_VEL
LIN {X 0,Y 377.661,Z 383.996,A -85,B 0,C 180,E1 17063.438,E2 17063.438} C_VEL
LIN {X 0,Y 377.672,Z 383.989,A -85,B 0,C 180,E1 17059.439,E2 17059.439} C_VEL
LIN {X 0,Y 377.675,Z 383.993,A -85,B 0,C 180,E1 17055.402,E2 17055.402} C_VEL
LIN {X 0,Y 377.689,Z 384.003,A -85,B 0,C 180,E1 17051.432,E2 17051.432} C_VEL
LIN {X 0,Y 377.737,Z 384.447,A -85,B 0,C 180,E1 17050.422,E2 17050.422} C_VEL
LIN {X 0,Y 378.305,Z 386.225,A -85,B 0,C 180,E1 17049.903,E2 17049.903} C_VEL
LIN {X 0,Y 380.339,Z 389.028,A -85,B 0,C 180,E1 17049.028,E2 17049.028} C_VEL
LIN {X 0,Y 383.308,Z 391.143,A -85,B 0,C 180,E1 17047.901,E2 17047.901} C_VEL
LIN {X 0,Y 385.423,Z 394.69,A -85,B 0,C 180,E1 17047.026,E2 17047.026} C_VEL
LIN {X 0,Y 388.682,Z 397.42,A -85,B 0,C 180,E1 17045.872,E2 17045.872} C_VEL
LIN {X 0,Y 391.33,Z 401.3,A -85,B 0,C 180,E1 17044.898,E2 17044.898} C_VEL
LIN {X 0,Y 393.933,Z 403.685,A -85,B 0,C 180,E1 17044.033,E2 17044.033} C_VEL
LIN {X 0,Y 397.151,Z 407.893,A -85,B 0,C 180,E1 17042.964,E2 17042.964} C_VEL
LIN {X 0,Y 399.146,Z 409.903,A -85,B 0,C 180,E1 17042.348,E2 17042.348} C_VEL
LIN {X 0,Y 402.787,Z 414.387,A -85,B 0,C 180,E1 17041.221,E2 17041.221} C_VEL
LIN {X 0,Y 409.344,Z 422.673,A -85,B 0,C 180,E1 17039.307,E2 17039.307} C_VEL
LIN {X 0,Y 414.47,Z 429.109,A -85,B 0,C 180,E1 17037.92,E2 17037.92} C_VEL
LIN {X 0,Y 424.635,Z 442.354,A -85,B 0,C 180,E1 17035.357,E2 17035.357} C_VEL
LIN {X 0,Y 437.256,Z 459.967,A -85,B 0,C 180,E1 17032.471,E2 17032.471} C_VEL
LIN {X 0,Y 440.296,Z 464.851,A -85,B 0,C 180,E1 17031.804,E2 17031.804} C_VEL
LIN {X 0,Y 430.654,Z 672.805,A -85,B 0,C 180,E1 17027.851,E2 17027.851} C_VEL
LIN {X 0,Y 428.865,Z 710.76,A -85,B 0,C 180,E1 17027.118,E2 17027.118} C_VEL
LIN {X 0,Y 427.395,Z 719.495,A -85,B 0,C 180,E1 17027.052,E2 17027.052} C_VEL
LIN {X 0,Y 422.094,Z 736.582,A -85,B 0,C 180,E1 17027.126,E2 17027.126} C_VEL
LIN {X 0,Y 420.504,Z 744.107,A -85,B 0,C 180,E1 17026.996,E2 17026.996} C_VEL
LIN {X 0,Y 420.381,Z 745.179,A -85,B 0,C 180,E1 17026.961,E2 17026.961} C_VEL
LIN {X 0,Y 417.517,Z 766.467,A -85,B 0,C 180,E1 17026.088,E2 17026.088} C_VEL
LIN {X 0,Y 414.239,Z 787.055,A -85,B 0,C 180,E1 17025.035,E2 17025.035} C_VEL
LIN {X 0,Y 410.364,Z 807.491,A -85,B 0,C 180,E1 17023.738,E2 17023.738} C_VEL
LIN {X 0,Y 406.143,Z 827.528,A -85,B 0,C 180,E1 17022.219,E2 17022.219} C_VEL
LIN {X 0,Y 401.427,Z 847.371,A -85,B 0,C 180,E1 17020.399,E2 17020.399} C_VEL
LIN {X 0,Y 396.616,Z 866.48,A -85,B 0,C 180,E1 17018.331,E2 17018.331} C_VEL
LIN {X 0,Y 392.038,Z 883.485,A -85,B 0,C 180,E1 17016.145,E2 17016.145} C_VEL
LIN {X 0,Y 387.242,Z 900.751,A -85,B 0,C 180,E1 17013.549,E2 17013.549} C_VEL
LIN {X 0,Y 383.271,Z 914.98,A -85,B 0,C 180,E1 17011.042,E2 17011.042} C_VEL
LIN {X 0,Y 379.184,Z 929.773,A -85,B 0,C 180,E1 17007.984,E2 17007.984} C_VEL
LIN {X 0,Y 375.939,Z 942.237,A -85,B 0,C 180,E1 17004.961,E2 17004.961} C_VEL
LIN {X 0,Y 373.156,Z 953.548,A -85,B 0,C 180,E1 17001.677,E2 17001.677} C_VEL
LIN {X 0,Y 371.084,Z 963.277,A -85,B 0,C 180,E1 16998.338,E2 16998.338} C_VEL
LIN {X 0,Y 369.614,Z 971.293,A -85,B 0,C 180,E1 16994.944,E2 16994.944} C_VEL
LIN {X 0,Y 368.647,Z 978.169,A -85,B 0,C 180,E1 16991.331,E2 16991.331} C_VEL
LIN {X 0,Y 368.205,Z 982.757,A -85,B 0,C 180,E1 16988.156,E2 16988.156} C_VEL
LIN {X 0,Y 367.989,Z 986.49,A -85,B 0,C 180,E1 16984.573,E2 16984.573} C_VEL
LIN {X 0,Y 367.943,Z 988.417,A -85,B 0,C 180,E1 16981.371,E2 16981.371} C_VEL
LIN {X 0,Y 367.927,Z 989.22,A -85,B 0,C 180,E1 16977.982,E2 16977.982} C_VEL
LIN {X 0,Y 367.94,Z 988.478,A -85,B 0,C 180,E1 16974.611,E2 16974.611} C_VEL
LIN {X 0,Y 367.998,Z 986.541,A -85,B 0,C 180,E1 16971.32,E2 16971.32} C_VEL
LIN {X 0,Y 368.207,Z 982.972,A -85,B 0,C 180,E1 16967.845,E2 16967.845} C_VEL
LIN {X 0,Y 368.652,Z 978.38,A -85,B 0,C 180,E1 16964.625,E2 16964.625} C_VEL
LIN {X 0,Y 369.627,Z 971.549,A -85,B 0,C 180,E1 16960.996,E2 16960.996} C_VEL
LIN {X 0,Y 371.042,Z 963.869,A -85,B 0,C 180,E1 16957.713,E2 16957.713} C_VEL
LIN {X 0,Y 373.107,Z 954.28,A -85,B 0,C 180,E1 16954.369,E2 16954.369} C_VEL
LIN {X 0,Y 375.896,Z 943.074,A -85,B 0,C 180,E1 16951.067,E2 16951.067} C_VEL
LIN {X 0,Y 379.234,Z 930.401,A -85,B 0,C 180,E1 16947.96,E2 16947.96} C_VEL
LIN {X 0,Y 383.318,Z 915.874,A -85,B 0,C 180,E1 16944.925,E2 16944.925} C_VEL
LIN {X 0,Y 387.277,Z 901.915,A -85,B 0,C 180,E1 16942.436,E2 16942.436} C_VEL
LIN {X 0,Y 392.284,Z 884.221,A -85,B 0,C 180,E1 16939.746,E2 16939.746} C_VEL
LIN {X 0,Y 396.834,Z 867.679,A -85,B 0,C 180,E1 16937.599,E2 16937.599} C_VEL
LIN {X 0,Y 401.653,Z 848.997,A -85,B 0,C 180,E1 16935.547,E2 16935.547} C_VEL
LIN {X 0,Y 406.409,Z 829.578,A -85,B 0,C 180,E1 16933.734,E2 16933.734} C_VEL
LIN {X 0,Y 410.607,Z 810.153,A -85,B 0,C 180,E1 16932.231,E2 16932.231} C_VEL
LIN {X 0,Y 414.678,Z 789.568,A -85,B 0,C 180,E1 16930.892,E2 16930.892} C_VEL
LIN {X 0,Y 418.069,Z 768.933,A -85,B 0,C 180,E1 16929.813,E2 16929.813} C_VEL
LIN {X 0,Y 421.116,Z 747.14,A -85,B 0,C 180,E1 16928.899,E2 16928.899} C_VEL
LIN {X 0,Y 423.372,Z 725.598,A -85,B 0,C 180,E1 16928.227,E2 16928.227} C_VEL
LIN {X 0,Y 425.142,Z 700.471,A -85,B 0,C 180,E1 16927.658,E2 16927.658} C_VEL
LIN {X 0,Y 435.523,Z 510.211,A -85,B 0,C 180,E1 16923.913,E2 16923.913} C_VEL
LIN {X 0,Y 437.891,Z 469.326,A -85,B 0,C 180,E1 16923.076,E2 16923.076} C_VEL
LIN {X 0,Y 430.597,Z 457.982,A -85,B 0,C 180,E1 16921.032,E2 16921.032} C_VEL
LIN {X 0,Y 424.677,Z 449.305,A -85,B 0,C 180,E1 16919.157,E2 16919.157} C_VEL
LIN {X 0,Y 419.335,Z 441.594,A -85,B 0,C 180,E1 16917.206,E2 16917.206} C_VEL
LIN {X 0,Y 415.239,Z 436.162,A -85,B 0,C 180,E1 16915.489,E2 16915.489} C_VEL
LIN {X 0,Y 411.969,Z 431.511,A -85,B 0,C 180,E1 16913.87,E2 16913.87} C_VEL
LIN {X 0,Y 408.531,Z 427.508,A -85,B 0,C 180,E1 16911.84,E2 16911.84} C_VEL
LIN {X 0,Y 407.574,Z 425.652,A -85,B 0,C 180,E1 16911.11,E2 16911.11} C_VEL
LIN {X 0,Y 404.276,Z 422.4,A -85,B 0,C 180,E1 16908.01,E2 16908.01} C_VEL
LIN {X 0,Y 403.384,Z 420.027,A -85,B 0,C 180,E1 16906.088,E2 16906.088} C_VEL
LIN {X 0,Y 403.185,Z 419.852,A -85,B 0,C 180,E1 16902.985,E2 16902.985} C_VEL
LIN {X 0,Y 403.688,Z 420.849,A -85,B 0,C 180,E1 16901.517,E2 16901.517} C_VEL
LIN {X 0,Y 405.736,Z 424.332,A -85,B 0,C 180,E1 16898.762,E2 16898.762} C_VEL
LIN {X 0,Y 407.77,Z 426.02,A -85,B 0,C 180,E1 16897.168,E2 16897.168} C_VEL
LIN {X 0,Y 410.575,Z 430.248,A -85,B 0,C 180,E1 16895.314,E2 16895.314} C_VEL
LIN {X 0,Y 412.219,Z 432.071,A -85,B 0,C 180,E1 16894.422,E2 16894.422} C_VEL
LIN {X 0,Y 416.193,Z 438.021,A -85,B 0,C 180,E1 16892.493,E2 16892.493} C_VEL
LIN {X 0,Y 420.892,Z 445.018,A -85,B 0,C 180,E1 16890.584,E2 16890.584} C_VEL
LIN {X 0,Y 428.158,Z 456.779,A -85,B 0,C 180,E1 16888.067,E2 16888.067} C_VEL
LIN {X 0,Y 435.264,Z 469.119,A -85,B 0,C 180,E1 16885.95,E2 16885.95} C_VEL
LIN {X 0,Y 437.895,Z 474.174,A -85,B 0,C 180,E1 16885.216,E2 16885.216} C_VEL
LIN {X 0,Y 427.609,Z 657.599,A -85,B 0,C 180,E1 16881.582,E2 16881.582} C_VEL
LIN {X 0,Y 423.427,Z 736.824,A -85,B 0,C 180,E1 16880.009,E2 16880.009} C_VEL
LIN {X 0,Y 420.964,Z 760.158,A -85,B 0,C 180,E1 16879.361,E2 16879.361} C_VEL
LIN {X 0,Y 417.974,Z 782.382,A -85,B 0,C 180,E1 16878.537,E2 16878.537} C_VEL
LIN {X 0,Y 414.42,Z 803.766,A -85,B 0,C 180,E1 16877.504,E2 16877.504} C_VEL
LIN {X 0,Y 410.221,Z 825.87,A -85,B 0,C 180,E1 16876.178,E2 16876.178} C_VEL
LIN {X 0,Y 405.897,Z 846.117,A -85,B 0,C 180,E1 16874.694,E2 16874.694} C_VEL
LIN {X 0,Y 400.93,Z 867.415,A -85,B 0,C 180,E1 16872.814,E2 16872.814} C_VEL
LIN {X 0,Y 396.101,Z 886.896,A -85,B 0,C 180,E1 16870.776,E2 16870.776} C_VEL
LIN {X 0,Y 391.249,Z 905.274,A -85,B 0,C 180,E1 16868.486,E2 16868.486} C_VEL
LIN {X 0,Y 386.509,Z 923.208,A -85,B 0,C 180,E1 16865.872,E2 16865.872} C_VEL
LIN {X 0,Y 382.486,Z 938.275,A -85,B 0,C 180,E1 16863.299,E2 16863.299} C_VEL
LIN {X 0,Y 378.418,Z 954.101,A -85,B 0,C 180,E1 16860.137,E2 16860.137} C_VEL
LIN {X 0,Y 375.297,Z 967.063,A -85,B 0,C 180,E1 16857.105,E2 16857.105} C_VEL
LIN {X 0,Y 372.653,Z 978.934,A -85,B 0,C 180,E1 16853.806,E2 16853.806} C_VEL
LIN {X 0,Y 370.746,Z 988.995,A -85,B 0,C 180,E1 16850.527,E2 16850.527} C_VEL
LIN {X 0,Y 369.402,Z 997.409,A -85,B 0,C 180,E1 16847.163,E2 16847.163} C_VEL
LIN {X 0,Y 368.578,Z 1004.364,A -85,B 0,C 180,E1 16843.796,E2 16843.796} C_VEL
LIN {X 0,Y 368.134,Z 1009.541,A -85,B 0,C 180,E1 16840.488,E2 16840.488} C_VEL
LIN {X 0,Y 367.959,Z 1013.076,A -85,B 0,C 180,E1 16837.498,E2 16837.498} C_VEL
LIN {X 0,Y 367.927,Z 1015.668,A -85,B 0,C 180,E1 16834.056,E2 16834.056} C_VEL
LIN {X 0,Y 367.917,Z 1016.651,A -85,B 0,C 180,E1 16831.094,E2 16831.094} C_VEL
LIN {X 0,Y 367.928,Z 1016.526,A -85,B 0,C 180,E1 16827.98,E2 16827.98} C_VEL
LIN {X 0,Y 367.93,Z 1014.833,A -85,B 0,C 180,E1 16824.546,E2 16824.546} C_VEL
LIN {X 0,Y 368.028,Z 1012.002,A -85,B 0,C 180,E1 16821.411,E2 16821.411} C_VEL
LIN {X 0,Y 368.335,Z 1007.064,A -85,B 0,C 180,E1 16817.748,E2 16817.748} C_VEL
LIN {X 0,Y 368.921,Z 1001.4,A -85,B 0,C 180,E1 16814.602,E2 16814.602} C_VEL
LIN {X 0,Y 370.12,Z 993.054,A -85,B 0,C 180,E1 16810.926,E2 16810.926} C_VEL
LIN {X 0,Y 371.731,Z 984.127,A -85,B 0,C 180,E1 16807.707,E2 16807.707} C_VEL
LIN {X 0,Y 374.092,Z 972.94,A -85,B 0,C 180,E1 16804.348,E2 16804.348} C_VEL
LIN {X 0,Y 377.097,Z 960.43,A -85,B 0,C 180,E1 16801.153,E2 16801.153} C_VEL
LIN {X 0,Y 380.632,Z 946.387,A -85,B 0,C 180,E1 16798.136,E2 16798.136} C_VEL
LIN {X 0,Y 384.706,Z 931.117,A -85,B 0,C 180,E1 16795.313,E2 16795.313} C_VEL
LIN {X 0,Y 388.895,Z 915.395,A -85,B 0,C 180,E1 16792.836,E2 16792.836} C_VEL
LIN {X 0,Y 394,Z 896.171,A -85,B 0,C 180,E1 16790.252,E2 16790.252} C_VEL
LIN {X 0,Y 398.505,Z 878.521,A -85,B 0,C 180,E1 16788.237,E2 16788.237} C_VEL
LIN {X 0,Y 403.297,Z 858.49,A -85,B 0,C 180,E1 16786.307,E2 16786.307} C_VEL
LIN {X 0,Y 407.782,Z 838.548,A -85,B 0,C 180,E1 16784.686,E2 16784.686} C_VEL
LIN {X 0,Y 411.961,Z 817.419,A -85,B 0,C 180,E1 16783.278,E2 16783.278} C_VEL
LIN {X 0,Y 415.703,Z 796.268,A -85,B 0,C 180,E1 16782.115,E2 16782.115} C_VEL
LIN {X 0,Y 418.863,Z 774.438,A -85,B 0,C 180,E1 16781.177,E2 16781.177} C_VEL
LIN {X 0,Y 421.543,Z 751.928,A -85,B 0,C 180,E1 16780.435,E2 16780.435} C_VEL
LIN {X 0,Y 423.338,Z 729.119,A -85,B 0,C 180,E1 16779.896,E2 16779.896} C_VEL
LIN {X 0,Y 433.344,Z 518.886,A -85,B 0,C 180,E1 16775.864,E2 16775.864} C_VEL
LIN {X 0,Y 435.473,Z 473.676,A -85,B 0,C 180,E1 16774.963,E2 16774.963} C_VEL
LIN {X 0,Y 425.477,Z 457.916,A -85,B 0,C 180,E1 16772.637,E2 16772.637} C_VEL
LIN {X 0,Y 415.962,Z 443.915,A -85,B 0,C 180,E1 16770.237,E2 16770.237} C_VEL
LIN {X 0,Y 405.735,Z 429.659,A -85,B 0,C 180,E1 16767.4,E2 16767.4} C_VEL
LIN {X 0,Y 397.908,Z 419.341,A -85,B 0,C 180,E1 16765.009,E2 16765.009} C_VEL
LIN {X 0,Y 393.237,Z 413.539,A -85,B 0,C 180,E1 16763.488,E2 16763.488} C_VEL
LIN {X 0,Y 390.44,Z 409.888,A -85,B 0,C 180,E1 16762.51,E2 16762.51} C_VEL
LIN {X 0,Y 387.083,Z 406.078,A -85,B 0,C 180,E1 16761.319,E2 16761.319} C_VEL
LIN {X 0,Y 385.715,Z 404.173,A -85,B 0,C 180,E1 16760.801,E2 16760.801} C_VEL
LIN {X 0,Y 382.477,Z 401.069,A -85,B 0,C 180,E1 16759.588,E2 16759.588} C_VEL
LIN {X 0,Y 380.737,Z 398.118,A -85,B 0,C 180,E1 16758.845,E2 16758.845} C_VEL
LIN {X 0,Y 377.503,Z 395.638,A -85,B 0,C 180,E1 16757.574,E2 16757.574} C_VEL
LIN {X 0,Y 375.018,Z 391.615,A -85,B 0,C 180,E1 16756.416,E2 16756.416} C_VEL
LIN {X 0,Y 371.681,Z 389.354,A -85,B 0,C 180,E1 16754.966,E2 16754.966} C_VEL
LIN {X 0,Y 370.013,Z 386.452,A -85,B 0,C 180,E1 16754.075,E2 16754.075} C_VEL
LIN {X 0,Y 369.739,Z 385.099,A -85,B 0,C 180,E1 16753.428,E2 16753.428} C_VEL
LIN {X 0,Y 369.721,Z 384.992,A -85,B 0,C 180,E1 16749.255,E2 16749.255} C_VEL
LIN {X 0,Y 369.727,Z 384.981,A -85,B 0,C 180,E1 16745.275,E2 16745.275} C_VEL
LIN {X 0,Y 369.733,Z 384.977,A -85,B 0,C 180,E1 16741.084,E2 16741.084} C_VEL
LIN {X 0,Y 369.729,Z 384.98,A -85,B 0,C 180,E1 16737.054,E2 16737.054} C_VEL
LIN {X 0,Y 369.745,Z 384.987,A -85,B 0,C 180,E1 16732.854,E2 16732.854} C_VEL
LIN {X 0,Y 369.737,Z 384.993,A -85,B 0,C 180,E1 16728.772,E2 16728.772} C_VEL
LIN {X 0,Y 369.747,Z 384.984,A -85,B 0,C 180,E1 16724.632,E2 16724.632} C_VEL
LIN {X 0,Y 369.74,Z 384.977,A -85,B 0,C 180,E1 16720.407,E2 16720.407} C_VEL
LIN {X 0,Y 369.746,Z 384.975,A -85,B 0,C 180,E1 16716.408,E2 16716.408} C_VEL
LIN {X 0,Y 369.748,Z 384.977,A -85,B 0,C 180,E1 16712.282,E2 16712.282} C_VEL
LIN {X 0,Y 369.751,Z 384.984,A -85,B 0,C 180,E1 16708.176,E2 16708.176} C_VEL
LIN {X 0,Y 369.745,Z 384.992,A -85,B 0,C 180,E1 16704.069,E2 16704.069} C_VEL
LIN {X 0,Y 369.752,Z 384.978,A -85,B 0,C 180,E1 16699.922,E2 16699.922} C_VEL
LIN {X 0,Y 369.745,Z 384.978,A -85,B 0,C 180,E1 16695.758,E2 16695.758} C_VEL
LIN {X 0,Y 369.765,Z 385.122,A -85,B 0,C 180,E1 16693.781,E2 16693.781} C_VEL
LIN {X 0,Y 370.056,Z 386.457,A -85,B 0,C 180,E1 16693.154,E2 16693.154} C_VEL
LIN {X 0,Y 371.694,Z 389.311,A -85,B 0,C 180,E1 16692.289,E2 16692.289} C_VEL
LIN {X 0,Y 375.547,Z 392.208,A -85,B 0,C 180,E1 16690.613,E2 16690.613} C_VEL
LIN {X 0,Y 377.639,Z 395.745,A -85,B 0,C 180,E1 16689.642,E2 16689.642} C_VEL
LIN {X 0,Y 381.031,Z 398.453,A -85,B 0,C 180,E1 16688.315,E2 16688.315} C_VEL
LIN {X 0,Y 383.559,Z 402.337,A -85,B 0,C 180,E1 16687.27,E2 16687.27} C_VEL
LIN {X 0,Y 386.422,Z 404.894,A -85,B 0,C 180,E1 16686.23,E2 16686.23} C_VEL
LIN {X 0,Y 389.552,Z 409.065,A -85,B 0,C 180,E1 16685.089,E2 16685.089} C_VEL
LIN {X 0,Y 391.645,Z 411.136,A -85,B 0,C 180,E1 16684.375,E2 16684.375} C_VEL
LIN {X 0,Y 395.178,Z 415.517,A -85,B 0,C 180,E1 16683.191,E2 16683.191} C_VEL
LIN {X 0,Y 396.849,Z 417.402,A -85,B 0,C 180,E1 16682.662,E2 16682.662} C_VEL
LIN {X 0,Y 401.792,Z 423.593,A -85,B 0,C 180,E1 16681.124,E2 16681.124} C_VEL
LIN {X 0,Y 407.146,Z 430.348,A -85,B 0,C 180,E1 16679.553,E2 16679.553} C_VEL
LIN {X 0,Y 413.781,Z 438.724,A -85,B 0,C 180,E1 16677.747,E2 16677.747} C_VEL
LIN {X 0,Y 424.833,Z 453.658,A -85,B 0,C 180,E1 16674.969,E2 16674.969} C_VEL
LIN {X 0,Y 435.291,Z 468.679,A -85,B 0,C 180,E1 16672.572,E2 16672.572} C_VEL
LIN {X 0,Y 425.265,Z 675.601,A -85,B 0,C 180,E1 16668.608,E2 16668.608} C_VEL
LIN {X 0,Y 423.037,Z 718.137,A -85,B 0,C 180,E1 16667.762,E2 16667.762} C_VEL
LIN {X 0,Y 420.829,Z 740.733,A -85,B 0,C 180,E1 16667.112,E2 16667.112} C_VEL
LIN {X 0,Y 420.381,Z 745.179,A -85,B 0,C 180,E1 16666.961,E2 16666.961} C_VEL
LIN {X 0,Y 418.865,Z 752.696,A -85,B 0,C 180,E1 16666.789,E2 16666.789} C_VEL
LIN {X 0,Y 411.989,Z 771.558,A -85,B 0,C 180,E1 16666.576,E2 16666.576} C_VEL
LIN {X 0,Y 410.057,Z 778.792,A -85,B 0,C 180,E1 16666.306,E2 16666.306} C_VEL
LIN {X 0,Y 406.336,Z 799.207,A -85,B 0,C 180,E1 16665.115,E2 16665.115} C_VEL
LIN {X 0,Y 401.843,Z 820.485,A -85,B 0,C 180,E1 16663.595,E2 16663.595} C_VEL
LIN {X 0,Y 397.248,Z 840.156,A -85,B 0,C 180,E1 16661.907,E2 16661.907} C_VEL
LIN {X 0,Y 392.368,Z 858.952,A -85,B 0,C 180,E1 16659.974,E2 16659.974} C_VEL
LIN {X 0,Y 387.402,Z 877.172,A -85,B 0,C 180,E1 16657.783,E2 16657.783} C_VEL
LIN {X 0,Y 382.578,Z 893.861,A -85,B 0,C 180,E1 16655.395,E2 16655.395} C_VEL
LIN {X 0,Y 377.662,Z 910.636,A -85,B 0,C 180,E1 16652.576,E2 16652.576} C_VEL
LIN {X 0,Y 373.61,Z 924.46,A -85,B 0,C 180,E1 16649.843,E2 16649.843} C_VEL
LIN {X 0,Y 369.803,Z 937.813,A -85,B 0,C 180,E1 16646.741,E2 16646.741} C_VEL
LIN {X 0,Y 366.721,Z 949.386,A -85,B 0,C 180,E1 16643.578,E2 16643.578} C_VEL
LIN {X 0,Y 364.19,Z 959.693,A -85,B 0,C 180,E1 16640.196,E2 16640.196} C_VEL
LIN {X 0,Y 362.367,Z 968.494,A -85,B 0,C 180,E1 16636.757,E2 16636.757} C_VEL
LIN {X 0,Y 361.14,Z 975.602,A -85,B 0,C 180,E1 16633.262,E2 16633.262} C_VEL
LIN {X 0,Y 360.409,Z 981.389,A -85,B 0,C 180,E1 16629.706,E2 16629.706} C_VEL
LIN {X 0,Y 360.067,Z 985.384,A -85,B 0,C 180,E1 16626.253,E2 16626.253} C_VEL
LIN {X 0,Y 359.953,Z 987.927,A -85,B 0,C 180,E1 16623.075,E2 16623.075} C_VEL
LIN {X 0,Y 359.917,Z 989.284,A -85,B 0,C 180,E1 16619.625,E2 16619.625} C_VEL
LIN {X 0,Y 359.925,Z 989.347,A -85,B 0,C 180,E1 16616.627,E2 16616.627} C_VEL
LIN {X 0,Y 359.94,Z 988.29,A -85,B 0,C 180,E1 16613.324,E2 16613.324} C_VEL
LIN {X 0,Y 360.071,Z 985.701,A -85,B 0,C 180,E1 16609.889,E2 16609.889} C_VEL
LIN {X 0,Y 360.363,Z 982.055,A -85,B 0,C 180,E1 16606.631,E2 16606.631} C_VEL
LIN {X 0,Y 361.086,Z 976.316,A -85,B 0,C 180,E1 16602.937,E2 16602.937} C_VEL
LIN {X 0,Y 362.24,Z 969.558,A -85,B 0,C 180,E1 16599.529,E2 16599.529} C_VEL
LIN {X 0,Y 364.064,Z 960.789,A -85,B 0,C 180,E1 16595.996,E2 16595.996} C_VEL
LIN {X 0,Y 366.599,Z 950.585,A -85,B 0,C 180,E1 16592.562,E2 16592.562} C_VEL
LIN {X 0,Y 369.748,Z 938.849,A -85,B 0,C 180,E1 16589.305,E2 16589.305} C_VEL
LIN {X 0,Y 373.823,Z 924.83,A -85,B 0,C 180,E1 16586.008,E2 16586.008} C_VEL
LIN {X 0,Y 378.047,Z 910.757,A -85,B 0,C 180,E1 16583.209,E2 16583.209} C_VEL
LIN {X 0,Y 382.87,Z 894.627,A -85,B 0,C 180,E1 16580.484,E2 16580.484} C_VEL
LIN {X 0,Y 387.961,Z 877.444,A -85,B 0,C 180,E1 16578.006,E2 16578.006} C_VEL
LIN {X 0,Y 392.916,Z 859.722,A -85,B 0,C 180,E1 16575.86,E2 16575.86} C_VEL
LIN {X 0,Y 397.999,Z 840.559,A -85,B 0,C 180,E1 16573.882,E2 16573.882} C_VEL
LIN {X 0,Y 402.504,Z 821.868,A -85,B 0,C 180,E1 16572.263,E2 16572.263} C_VEL
LIN {X 0,Y 407.228,Z 800.09,A -85,B 0,C 180,E1 16570.691,E2 16570.691} C_VEL
LIN {X 0,Y 411.222,Z 778.921,A -85,B 0,C 180,E1 16569.447,E2 16569.447} C_VEL
LIN {X 0,Y 414.746,Z 756.365,A -85,B 0,C 180,E1 16568.4,E2 16568.4} C_VEL
LIN {X 0,Y 417.626,Z 733.557,A -85,B 0,C 180,E1 16567.586,E2 16567.586} C_VEL
LIN {X 0,Y 419.587,Z 710.568,A -85,B 0,C 180,E1 16567.009,E2 16567.009} C_VEL
LIN {X 0,Y 431.35,Z 508.105,A -85,B 0,C 180,E1 16562.973,E2 16562.973} C_VEL
LIN {X 0,Y 433.529,Z 473.789,A -85,B 0,C 180,E1 16562.281,E2 16562.281} C_VEL
LIN {X 0,Y 426.107,Z 462.06,A -85,B 0,C 180,E1 16560.061,E2 16560.061} C_VEL
LIN {X 0,Y 419.717,Z 452.634,A -85,B 0,C 180,E1 16557.85,E2 16557.85} C_VEL
LIN {X 0,Y 416.273,Z 447.802,A -85,B 0,C 180,E1 16556.489,E2 16556.489} C_VEL
LIN {X 0,Y 413.267,Z 443.531,A -85,B 0,C 180,E1 16555.143,E2 16555.143} C_VEL
LIN {X 0,Y 409.744,Z 438.624,A -85,B 0,C 180,E1 16553.31,E2 16553.31} C_VEL
LIN {X 0,Y 406.626,Z 434.469,A -85,B 0,C 180,E1 16551.307,E2 16551.307} C_VEL
LIN {X 0,Y 405.99,Z 433.343,A -85,B 0,C 180,E1 16550.789,E2 16550.789} C_VEL
LIN {X 0,Y 402.934,Z 429.991,A -85,B 0,C 180,E1 16547.679,E2 16547.679} C_VEL
LIN {X 0,Y 402.207,Z 427.88,A -85,B 0,C 180,E1 16545.9,E2 16545.9} C_VEL
LIN {X 0,Y 402.116,Z 427.809,A -85,B 0,C 180,E1 16542.789,E2 16542.789} C_VEL
LIN {X 0,Y 402.574,Z 428.967,A -85,B 0,C 180,E1 16541.464,E2 16541.464} C_VEL
LIN {X 0,Y 404.672,Z 432.373,A -85,B 0,C 180,E1 16538.703,E2 16538.703} C_VEL
LIN {X 0,Y 406.268,Z 433.72,A -85,B 0,C 180,E1 16537.423,E2 16537.423} C_VEL
LIN {X 0,Y 409.046,Z 437.956,A -85,B 0,C 180,E1 16535.524,E2 16535.524} C_VEL
LIN {X 0,Y 410.452,Z 439.588,A -85,B 0,C 180,E1 16534.729,E2 16534.729} C_VEL
LIN {X 0,Y 415.446,Z 447.109,A -85,B 0,C 180,E1 16532.284,E2 16532.284} C_VEL
LIN {X 0,Y 421.096,Z 456.335,A -85,B 0,C 180,E1 16530.013,E2 16530.013} C_VEL
LIN {X 0,Y 427.942,Z 467.937,A -85,B 0,C 180,E1 16527.693,E2 16527.693} C_VEL
LIN {X 0,Y 433.459,Z 478.185,A -85,B 0,C 180,E1 16526.038,E2 16526.038} C_VEL
LIN {X 0,Y 422.641,Z 660.897,A -85,B 0,C 180,E1 16522.385,E2 16522.385} C_VEL
LIN {X 0,Y 418.379,Z 736.647,A -85,B 0,C 180,E1 16520.861,E2 16520.861} C_VEL
LIN {X 0,Y 415.817,Z 760.013,A -85,B 0,C 180,E1 16520.208,E2 16520.208} C_VEL
LIN {X 0,Y 412.676,Z 782.305,A -85,B 0,C 180,E1 16519.376,E2 16519.376} C_VEL
LIN {X 0,Y 409.079,Z 803.046,A -85,B 0,C 180,E1 16518.37,E2 16518.37} C_VEL
LIN {X 0,Y 404.606,Z 825.613,A -85,B 0,C 180,E1 16517.013,E2 16517.013} C_VEL
LIN {X 0,Y 400.087,Z 845.807,A -85,B 0,C 180,E1 16515.523,E2 16515.523} C_VEL
LIN {X 0,Y 394.889,Z 867.065,A -85,B 0,C 180,E1 16513.631,E2 16513.631} C_VEL
LIN {X 0,Y 389.94,Z 886.138,A -85,B 0,C 180,E1 16511.617,E2 16511.617} C_VEL
LIN {X 0,Y 384.895,Z 904.319,A -85,B 0,C 180,E1 16509.338,E2 16509.338} C_VEL
LIN {X 0,Y 380.159,Z 921.389,A -85,B 0,C 180,E1 16506.849,E2 16506.849} C_VEL
LIN {X 0,Y 375.702,Z 937.126,A -85,B 0,C 180,E1 16504.141,E2 16504.141} C_VEL
LIN {X 0,Y 371.57,Z 952.266,A -85,B 0,C 180,E1 16501.111,E2 16501.111} C_VEL
LIN {X 0,Y 368.157,Z 965.368,A -85,B 0,C 180,E1 16498.028,E2 16498.028} C_VEL
LIN {X 0,Y 365.213,Z 977.716,A -85,B 0,C 180,E1 16494.594,E2 16494.594} C_VEL
LIN {X 0,Y 363.148,Z 987.697,A -85,B 0,C 180,E1 16491.315,E2 16491.315} C_VEL
LIN {X 0,Y 361.632,Z 996.325,A -85,B 0,C 180,E1 16487.876,E2 16487.876} C_VEL
LIN {X 0,Y 360.726,Z 1003.065,A -85,B 0,C 180,E1 16484.613,E2 16484.613} C_VEL
LIN {X 0,Y 360.192,Z 1008.788,A -85,B 0,C 180,E1 16481.046,E2 16481.046} C_VEL
LIN {X 0,Y 360.001,Z 1012.429,A -85,B 0,C 180,E1 16477.986,E2 16477.986} C_VEL
LIN {X 0,Y 359.927,Z 1015.22,A -85,B 0,C 180,E1 16474.465,E2 16474.465} C_VEL
LIN {X 0,Y 359.929,Z 1016.327,A -85,B 0,C 180,E1 16471.278,E2 16471.278} C_VEL
LIN {X 0,Y 359.932,Z 1016.274,A -85,B 0,C 180,E1 16468.253,E2 16468.253} C_VEL
LIN {X 0,Y 359.933,Z 1014.769,A -85,B 0,C 180,E1 16464.745,E2 16464.745} C_VEL
LIN {X 0,Y 360.026,Z 1012.032,A -85,B 0,C 180,E1 16461.54,E2 16461.54} C_VEL
LIN {X 0,Y 360.295,Z 1007.597,A -85,B 0,C 180,E1 16457.992,E2 16457.992} C_VEL
LIN {X 0,Y 360.923,Z 1001.715,A -85,B 0,C 180,E1 16454.582,E2 16454.582} C_VEL
LIN {X 0,Y 362.032,Z 994.395,A -85,B 0,C 180,E1 16451.153,E2 16451.153} C_VEL
LIN {X 0,Y 363.725,Z 985.235,A -85,B 0,C 180,E1 16447.712,E2 16447.712} C_VEL
LIN {X 0,Y 366.157,Z 974.355,A -85,B 0,C 180,E1 16444.273,E2 16444.273} C_VEL
LIN {X 0,Y 369.052,Z 962.672,A -85,B 0,C 180,E1 16441.173,E2 16441.173} C_VEL
LIN {X 0,Y 372.885,Z 948.272,A -85,B 0,C 180,E1 16437.921,E2 16437.921} C_VEL
LIN {X 0,Y 376.807,Z 934.266,A -85,B 0,C 180,E1 16435.221,E2 16435.221} C_VEL
LIN {X 0,Y 381.563,Z 917.341,A -85,B 0,C 180,E1 16432.436,E2 16432.436} C_VEL
LIN {X 0,Y 386.522,Z 899.754,A -85,B 0,C 180,E1 16429.968,E2 16429.968} C_VEL
LIN {X 0,Y 391.411,Z 881.365,A -85,B 0,C 180,E1 16427.798,E2 16427.798} C_VEL
LIN {X 0,Y 396.481,Z 861.451,A -85,B 0,C 180,E1 16425.798,E2 16425.798} C_VEL
LIN {X 0,Y 400.991,Z 842.214,A -85,B 0,C 180,E1 16424.183,E2 16424.183} C_VEL
LIN {X 0,Y 405.688,Z 820.055,A -85,B 0,C 180,E1 16422.643,E2 16422.643} C_VEL
LIN {X 0,Y 409.319,Z 800.5,A -85,B 0,C 180,E1 16421.53,E2 16421.53} C_VEL
LIN {X 0,Y 412.995,Z 777.135,A -85,B 0,C 180,E1 16420.473,E2 16420.473} C_VEL
LIN {X 0,Y 415.56,Z 757.199,A -85,B 0,C 180,E1 16419.779,E2 16419.779} C_VEL
LIN {X 0,Y 417.793,Z 732.729,A -85,B 0,C 180,E1 16419.154,E2 16419.154} C_VEL
LIN {X 0,Y 428.199,Z 524.376,A -85,B 0,C 180,E1 16415.12,E2 16415.12} C_VEL
LIN {X 0,Y 430.541,Z 477.753,A -85,B 0,C 180,E1 16414.194,E2 16414.194} C_VEL
LIN {X 0,Y 420.759,Z 462.325,A -85,B 0,C 180,E1 16411.839,E2 16411.839} C_VEL
LIN {X 0,Y 412.239,Z 449.638,A -85,B 0,C 180,E1 16409.615,E2 16409.615} C_VEL
LIN {X 0,Y 402.607,Z 436.085,A -85,B 0,C 180,E1 16406.871,E2 16406.871} C_VEL
LIN {X 0,Y 394.767,Z 425.71,A -85,B 0,C 180,E1 16404.423,E2 16404.423} C_VEL
LIN {X 0,Y 388.214,Z 417.235,A -85,B 0,C 180,E1 16402.167,E2 16402.167} C_VEL
LIN {X 0,Y 384.607,Z 413.043,A -85,B 0,C 180,E1 16400.864,E2 16400.864} C_VEL
LIN {X 0,Y 383.334,Z 411.434,A -85,B 0,C 180,E1 16400.377,E2 16400.377} C_VEL
LIN {X 0,Y 379.992,Z 407.912,A -85,B 0,C 180,E1 16399.082,E2 16399.082} C_VEL
LIN {X 0,Y 378.393,Z 405.503,A -85,B 0,C 180,E1 16398.406,E2 16398.406} C_VEL
LIN {X 0,Y 375.095,Z 402.532,A -85,B 0,C 180,E1 16397.05,E2 16397.05} C_VEL
LIN {X 0,Y 373.288,Z 399.338,A -85,B 0,C 180,E1 16396.174,E2 16396.174} C_VEL
LIN {X 0,Y 369.662,Z 396.673,A -85,B 0,C 180,E1 16394.568,E2 16394.568} C_VEL
LIN {X 0,Y 367.725,Z 393.258,A -85,B 0,C 180,E1 16393.523,E2 16393.523} C_VEL
LIN {X 0,Y 366.533,Z 392.355,A -85,B 0,C 180,E1 16392.925,E2 16392.925} C_VEL
LIN {X 0,Y 363.587,Z 390.118,A -85,B 0,C 180,E1 16391.419,E2 16391.419} C_VEL
LIN {X 0,Y 361.879,Z 386.741,A -85,B 0,C 180,E1 16390.185,E2 16390.185} C_VEL
LIN {X 0,Y 361.79,Z 386.019,A -85,B 0,C 180,E1 16389.384,E2 16389.384} C_VEL
LIN {X 0,Y 361.786,Z 385.969,A -85,B 0,C 180,E1 16385.232,E2 16385.232} C_VEL
LIN {X 0,Y 361.794,Z 385.965,A -85,B 0,C 180,E1 16381.108,E2 16381.108} C_VEL
LIN {X 0,Y 361.787,Z 385.97,A -85,B 0,C 180,E1 16376.932,E2 16376.932} C_VEL
LIN {X 0,Y 361.797,Z 385.978,A -85,B 0,C 180,E1 16372.757,E2 16372.757} C_VEL
LIN {X 0,Y 361.796,Z 385.982,A -85,B 0,C 180,E1 16368.684,E2 16368.684} C_VEL
LIN {X 0,Y 361.807,Z 385.972,A -85,B 0,C 180,E1 16364.615,E2 16364.615} C_VEL
LIN {X 0,Y 361.802,Z 385.965,A -85,B 0,C 180,E1 16360.436,E2 16360.436} C_VEL
LIN {X 0,Y 361.805,Z 385.964,A -85,B 0,C 180,E1 16356.377,E2 16356.377} C_VEL
LIN {X 0,Y 361.811,Z 385.966,A -85,B 0,C 180,E1 16352.154,E2 16352.154} C_VEL
LIN {X 0,Y 361.807,Z 385.975,A -85,B 0,C 180,E1 16348.027,E2 16348.027} C_VEL
LIN {X 0,Y 361.804,Z 385.978,A -85,B 0,C 180,E1 16343.939,E2 16343.939} C_VEL
LIN {X 0,Y 361.81,Z 385.965,A -85,B 0,C 180,E1 16339.709,E2 16339.709} C_VEL
LIN {X 0,Y 361.839,Z 386.309,A -85,B 0,C 180,E1 16337.301,E2 16337.301} C_VEL
LIN {X 0,Y 362.205,Z 387.719,A -85,B 0,C 180,E1 16336.687,E2 16336.687} C_VEL
LIN {X 0,Y 364.086,Z 390.639,A -85,B 0,C 180,E1 16335.55,E2 16335.55} C_VEL
LIN {X 0,Y 367.734,Z 393.15,A -85,B 0,C 180,E1 16333.733,E2 16333.733} C_VEL
LIN {X 0,Y 369.579,Z 396.513,A -85,B 0,C 180,E1 16332.733,E2 16332.733} C_VEL
LIN {X 0,Y 372.867,Z 399.096,A -85,B 0,C 180,E1 16331.267,E2 16331.267} C_VEL
LIN {X 0,Y 373.582,Z 399.919,A -85,B 0,C 180,E1 16330.944,E2 16330.944} C_VEL
LIN {X 0,Y 376.078,Z 403.649,A -85,B 0,C 180,E1 16329.794,E2 16329.794} C_VEL
LIN {X 0,Y 378.946,Z 406.091,A -85,B 0,C 180,E1 16328.647,E2 16328.647} C_VEL
LIN {X 0,Y 381.788,Z 410.057,A -85,B 0,C 180,E1 16327.484,E2 16327.484} C_VEL
LIN {X 0,Y 384.241,Z 412.391,A -85,B 0,C 180,E1 16326.57,E2 16326.57} C_VEL
LIN {X 0,Y 387.644,Z 416.693,A -85,B 0,C 180,E1 16325.323,E2 16325.323} C_VEL
LIN {X 0,Y 389.34,Z 418.481,A -85,B 0,C 180,E1 16324.735,E2 16324.735} C_VEL
LIN {X 0,Y 393.216,Z 423.137,A -85,B 0,C 180,E1 16323.418,E2 16323.418} C_VEL
LIN {X 0,Y 399.389,Z 430.947,A -85,B 0,C 180,E1 16321.453,E2 16321.453} C_VEL
LIN {X 0,Y 407.275,Z 440.85,A -85,B 0,C 180,E1 16319.147,E2 16319.147} C_VEL
LIN {X 0,Y 418.632,Z 456.102,A -85,B 0,C 180,E1 16316.137,E2 16316.137} C_VEL
LIN {X 0,Y 430.318,Z 472.773,A -85,B 0,C 180,E1 16313.351,E2 16313.351} C_VEL
LIN {X 0,Y 419.974,Z 677.399,A -85,B 0,C 180,E1 16309.402,E2 16309.402} C_VEL
LIN {X 0,Y 417.71,Z 718.582,A -85,B 0,C 180,E1 16308.574,E2 16308.574} C_VEL
LIN {X 0,Y 415.423,Z 741.144,A -85,B 0,C 180,E1 16307.921,E2 16307.921} C_VEL
LIN {X 0,Y 412.299,Z 764.817,A -85,B 0,C 180,E1 16306.987,E2 16306.987} C_VEL
LIN {X 0,Y 410.057,Z 778.792,A -85,B 0,C 180,E1 16306.306,E2 16306.306} C_VEL
LIN {X 0,Y 408.083,Z 786.227,A -85,B 0,C 180,E1 16306.009,E2 16306.009} C_VEL
LIN {X 0,Y 400.383,Z 804.442,A -85,B 0,C 180,E1 16305.505,E2 16305.505} C_VEL
LIN {X 0,Y 398.216,Z 811.184,A -85,B 0,C 180,E1 16305.129,E2 16305.129} C_VEL
LIN {X 0,Y 393.083,Z 833.036,A -85,B 0,C 180,E1 16303.379,E2 16303.379} C_VEL
LIN {X 0,Y 388.27,Z 851.72,A -85,B 0,C 180,E1 16301.583,E2 16301.583} C_VEL
LIN {X 0,Y 383.072,Z 870.243,A -85,B 0,C 180,E1 16299.46,E2 16299.46} C_VEL
LIN {X 0,Y 378.017,Z 887.554,A -85,B 0,C 180,E1 16297.137,E2 16297.137} C_VEL
LIN {X 0,Y 373.106,Z 903.438,A -85,B 0,C 180,E1 16294.607,E2 16294.607} C_VEL
LIN {X 0,Y 368.565,Z 918.302,A -85,B 0,C 180,E1 16291.861,E2 16291.861} C_VEL
LIN {X 0,Y 364.389,Z 931.812,A -85,B 0,C 180,E1 16288.895,E2 16288.895} C_VEL
LIN {X 0,Y 360.598,Z 944.82,A -85,B 0,C 180,E1 16285.543,E2 16285.543} C_VEL
LIN {X 0,Y 357.712,Z 955.416,A -85,B 0,C 180,E1 16282.286,E2 16282.286} C_VEL
LIN {X 0,Y 355.321,Z 965.281,A -85,B 0,C 180,E1 16278.636,E2 16278.636} C_VEL
LIN {X 0,Y 353.801,Z 972.78,A -85,B 0,C 180,E1 16275.261,E2 16275.261} C_VEL
LIN {X 0,Y 352.765,Z 979.151,A -85,B 0,C 180,E1 16271.659,E2 16271.659} C_VEL
LIN {X 0,Y 352.257,Z 983.67,A -85,B 0,C 180,E1 16268.342,E2 16268.342} C_VEL
LIN {X 0,Y 352.008,Z 987.266,A -85,B 0,C 180,E1 16264.591,E2 16264.591} C_VEL
LIN {X 0,Y 351.956,Z 989.1,A -85,B 0,C 180,E1 16261.304,E2 16261.304} C_VEL
LIN {X 0,Y 351.935,Z 989.793,A -85,B 0,C 180,E1 16257.712,E2 16257.712} C_VEL
LIN {X 0,Y 351.952,Z 989.037,A -85,B 0,C 180,E1 16254.341,E2 16254.341} C_VEL
LIN {X 0,Y 352.036,Z 987.035,A -85,B 0,C 180,E1 16250.84,E2 16250.84} C_VEL
LIN {X 0,Y 352.3,Z 983.468,A -85,B 0,C 180,E1 16247.285,E2 16247.285} C_VEL
LIN {X 0,Y 352.893,Z 978.711,A -85,B 0,C 180,E1 16243.824,E2 16243.824} C_VEL
LIN {X 0,Y 354.048,Z 971.875,A -85,B 0,C 180,E1 16240.083,E2 16240.083} C_VEL
LIN {X 0,Y 355.808,Z 963.813,A -85,B 0,C 180,E1 16236.512,E2 16236.512} C_VEL
LIN {X 0,Y 358.294,Z 953.868,A -85,B 0,C 180,E1 16232.968,E2 16232.968} C_VEL
LIN {X 0,Y 361.668,Z 942.046,A -85,B 0,C 180,E1 16229.439,E2 16229.439} C_VEL
LIN {X 0,Y 365.254,Z 930.222,A -85,B 0,C 180,E1 16226.468,E2 16226.468} C_VEL
LIN {X 0,Y 370.015,Z 915.031,A -85,B 0,C 180,E1 16223.237,E2 16223.237} C_VEL
LIN {X 0,Y 374.989,Z 899.54,A -85,B 0,C 180,E1 16220.445,E2 16220.445} C_VEL
LIN {X 0,Y 380.112,Z 882.915,A -85,B 0,C 180,E1 16217.925,E2 16217.925} C_VEL
LIN {X 0,Y 385.599,Z 864.657,A -85,B 0,C 180,E1 16215.568,E2 16215.568} C_VEL
LIN {X 0,Y 390.648,Z 846.736,A -85,B 0,C 180,E1 16213.62,E2 16213.62} C_VEL
LIN {X 0,Y 396.023,Z 826.005,A -85,B 0,C 180,E1 16211.727,E2 16211.727} C_VEL
LIN {X 0,Y 400.561,Z 806.644,A -85,B 0,C 180,E1 16210.252,E2 16210.252} C_VEL
LIN {X 0,Y 405.013,Z 784.691,A -85,B 0,C 180,E1 16208.883,E2 16208.883} C_VEL
LIN {X 0,Y 408.884,Z 762.426,A -85,B 0,C 180,E1 16207.768,E2 16207.768} C_VEL
LIN {X 0,Y 411.956,Z 739.777,A -85,B 0,C 180,E1 16206.904,E2 16206.904} C_VEL
LIN {X 0,Y 414.468,Z 714.845,A -85,B 0,C 180,E1 16206.22,E2 16206.22} C_VEL
LIN {X 0,Y 427.277,Z 507.108,A -85,B 0,C 180,E1 16202.034,E2 16202.034} C_VEL
LIN {X 0,Y 429.166,Z 478.137,A -85,B 0,C 180,E1 16201.432,E2 16201.432} C_VEL
LIN {X 0,Y 422.63,Z 467.701,A -85,B 0,C 180,E1 16199.357,E2 16199.357} C_VEL
LIN {X 0,Y 417.075,Z 459.258,A -85,B 0,C 180,E1 16197.321,E2 16197.321} C_VEL
LIN {X 0,Y 413.951,Z 454.743,A -85,B 0,C 180,E1 16196.02,E2 16196.02} C_VEL
LIN {X 0,Y 411.28,Z 450.844,A -85,B 0,C 180,E1 16194.77,E2 16194.77} C_VEL
LIN {X 0,Y 408.003,Z 446.154,A -85,B 0,C 180,E1 16192.992,E2 16192.992} C_VEL
LIN {X 0,Y 404.972,Z 441.78,A -85,B 0,C 180,E1 16190.909,E2 16190.909} C_VEL
LIN {X 0,Y 404.231,Z 440.896,A -85,B 0,C 180,E1 16190.317,E2 16190.317} C_VEL
LIN {X 0,Y 401.586,Z 437.474,A -85,B 0,C 180,E1 16187.271,E2 16187.271} C_VEL
LIN {X 0,Y 401.081,Z 435.798,A -85,B 0,C 180,E1 16185.86,E2 16185.86} C_VEL
LIN {X 0,Y 401.019,Z 435.742,A -85,B 0,C 180,E1 16182.739,E2 16182.739} C_VEL
LIN {X 0,Y 401.498,Z 437.226,A -85,B 0,C 180,E1 16181.337,E2 16181.337} C_VEL
LIN {X 0,Y 403.943,Z 440.692,A -85,B 0,C 180,E1 16178.358,E2 16178.358} C_VEL
LIN {X 0,Y 404.901,Z 441.693,A -85,B 0,C 180,E1 16177.573,E2 16177.573} C_VEL
LIN {X 0,Y 407.758,Z 445.904,A -85,B 0,C 180,E1 16175.596,E2 16175.596} C_VEL
LIN {X 0,Y 408.995,Z 447.639,A -85,B 0,C 180,E1 16174.865,E2 16174.865} C_VEL
LIN {X 0,Y 412.648,Z 453.353,A -85,B 0,C 180,E1 16172.98,E2 16172.98} C_VEL
LIN {X 0,Y 417.868,Z 461.93,A -85,B 0,C 180,E1 16170.744,E2 16170.744} C_VEL
LIN {X 0,Y 423.45,Z 471.732,A -85,B 0,C 180,E1 16168.704,E2 16168.704} C_VEL
LIN {X 0,Y 429.14,Z 482.152,A -85,B 0,C 180,E1 16166.883,E2 16166.883} C_VEL
LIN {X 0,Y 417.949,Z 661.193,A -85,B 0,C 180,E1 16163.269,E2 16163.269} C_VEL
LIN {X 0,Y 413.47,Z 736.542,A -85,B 0,C 180,E1 16161.737,E2 16161.737} C_VEL
LIN {X 0,Y 410.812,Z 759.739,A -85,B 0,C 180,E1 16161.084,E2 16161.084} C_VEL
LIN {X 0,Y 407.475,Z 782.307,A -85,B 0,C 180,E1 16160.236,E2 16160.236} C_VEL
LIN {X 0,Y 403.621,Z 803.614,A -85,B 0,C 180,E1 16159.195,E2 16159.195} C_VEL
LIN {X 0,Y 398.807,Z 826.636,A -85,B 0,C 180,E1 16157.786,E2 16157.786} C_VEL
LIN {X 0,Y 393.949,Z 847.367,A -85,B 0,C 180,E1 16156.229,E2 16156.229} C_VEL
LIN {X 0,Y 388.742,Z 867.511,A -85,B 0,C 180,E1 16154.398,E2 16154.398} C_VEL
LIN {X 0,Y 383.396,Z 887.108,A -85,B 0,C 180,E1 16152.29,E2 16152.29} C_VEL
LIN {X 0,Y 378.142,Z 905.099,A -85,B 0,C 180,E1 16149.984,E2 16149.984} C_VEL
LIN {X 0,Y 372.89,Z 922.916,A -85,B 0,C 180,E1 16147.304,E2 16147.304} C_VEL
LIN {X 0,Y 368.517,Z 937.651,A -85,B 0,C 180,E1 16144.706,E2 16144.706} C_VEL
LIN {X 0,Y 363.975,Z 953.333,A -85,B 0,C 180,E1 16141.466,E2 16141.466} C_VEL
LIN {X 0,Y 360.435,Z 966.304,A -85,B 0,C 180,E1 16138.321,E2 16138.321} C_VEL
LIN {X 0,Y 357.5,Z 977.882,A -85,B 0,C 180,E1 16134.985,E2 16134.985} C_VEL
LIN {X 0,Y 355.226,Z 988.276,A -85,B 0,C 180,E1 16131.467,E2 16131.467} C_VEL
LIN {X 0,Y 353.655,Z 996.712,A -85,B 0,C 180,E1 16127.953,E2 16127.953} C_VEL
LIN {X 0,Y 352.69,Z 1003.662,A -85,B 0,C 180,E1 16124.45,E2 16124.45} C_VEL
LIN {X 0,Y 352.184,Z 1008.895,A -85,B 0,C 180,E1 16120.969,E2 16120.969} C_VEL
LIN {X 0,Y 351.973,Z 1012.613,A -85,B 0,C 180,E1 16117.677,E2 16117.677} C_VEL
LIN {X 0,Y 351.936,Z 1015.131,A -85,B 0,C 180,E1 16114.077,E2 16114.077} C_VEL
LIN {X 0,Y 351.93,Z 1016.052,A -85,B 0,C 180,E1 16111.144,E2 16111.144} C_VEL
LIN {X 0,Y 351.938,Z 1015.93,A -85,B 0,C 180,E1 16107.888,E2 16107.888} C_VEL
LIN {X 0,Y 351.937,Z 1014.239,A -85,B 0,C 180,E1 16104.298,E2 16104.298} C_VEL
LIN {X 0,Y 352.044,Z 1011.404,A -85,B 0,C 180,E1 16101.018,E2 16101.018} C_VEL
LIN {X 0,Y 352.412,Z 1006.507,A -85,B 0,C 180,E1 16097.219,E2 16097.219} C_VEL
LIN {X 0,Y 353.108,Z 1000.777,A -85,B 0,C 180,E1 16093.894,E2 16093.894} C_VEL
LIN {X 0,Y 354.497,Z 992.405,A -85,B 0,C 180,E1 16090.05,E2 16090.05} C_VEL
LIN {X 0,Y 356.355,Z 983.487,A -85,B 0,C 180,E1 16086.701,E2 16086.701} C_VEL
LIN {X 0,Y 359.061,Z 972.23,A -85,B 0,C 180,E1 16083.191,E2 16083.191} C_VEL
LIN {X 0,Y 362.455,Z 959.678,A -85,B 0,C 180,E1 16079.87,E2 16079.87} C_VEL
LIN {X 0,Y 366.464,Z 945.574,A -85,B 0,C 180,E1 16076.748,E2 16076.748} C_VEL
LIN {X 0,Y 371.132,Z 929.758,A -85,B 0,C 180,E1 16073.754,E2 16073.754} C_VEL
LIN {X 0,Y 375.812,Z 913.964,A -85,B 0,C 180,E1 16071.217,E2 16071.217} C_VEL
LIN {X 0,Y 381.262,Z 895.101,A -85,B 0,C 180,E1 16068.641,E2 16068.641} C_VEL
LIN {X 0,Y 386.418,Z 876.711,A -85,B 0,C 180,E1 16066.514,E2 16066.514} C_VEL
LIN {X 0,Y 391.513,Z 857,A -85,B 0,C 180,E1 16064.611,E2 16064.611} C_VEL
LIN {X 0,Y 396.327,Z 837.095,A -85,B 0,C 180,E1 16062.986,E2 16062.986} C_VEL
LIN {X 0,Y 400.804,Z 815.911,A -85,B 0,C 180,E1 16061.572,E2 16061.572} C_VEL
LIN {X 0,Y 404.886,Z 794.066,A -85,B 0,C 180,E1 16060.382,E2 16060.382} C_VEL
LIN {X 0,Y 408.22,Z 772.508,A -85,B 0,C 180,E1 16059.461,E2 16059.461} C_VEL
LIN {X 0,Y 411.25,Z 747.738,A -85,B 0,C 180,E1 16058.675,E2 16058.675} C_VEL
LIN {X 0,Y 413.109,Z 724.325,A -85,B 0,C 180,E1 16058.136,E2 16058.136} C_VEL
LIN {X 0,Y 423.848,Z 516.476,A -85,B 0,C 180,E1 16054.099,E2 16054.099} C_VEL
LIN {X 0,Y 425.621,Z 481.584,A -85,B 0,C 180,E1 16053.387,E2 16053.387} C_VEL
LIN {X 0,Y 413.696,Z 462.879,A -85,B 0,C 180,E1 16050.38,E2 16050.38} C_VEL
LIN {X 0,Y 403.144,Z 447.568,A -85,B 0,C 180,E1 16047.431,E2 16047.431} C_VEL
LIN {X 0,Y 396.15,Z 438.009,A -85,B 0,C 180,E1 16045.288,E2 16045.288} C_VEL
LIN {X 0,Y 389.53,Z 429.127,A -85,B 0,C 180,E1 16043.084,E2 16043.084} C_VEL
LIN {X 0,Y 385.586,Z 424.213,A -85,B 0,C 180,E1 16041.685,E2 16041.685} C_VEL
LIN {X 0,Y 381.896,Z 419.581,A -85,B 0,C 180,E1 16040.297,E2 16040.297} C_VEL
LIN {X 0,Y 377.682,Z 414.997,A -85,B 0,C 180,E1 16038.642,E2 16038.642} C_VEL
LIN {X 0,Y 376.257,Z 412.939,A -85,B 0,C 180,E1 16038.034,E2 16038.034} C_VEL
LIN {X 0,Y 372.877,Z 409.627,A -85,B 0,C 180,E1 16036.593,E2 16036.593} C_VEL
LIN {X 0,Y 371.208,Z 406.839,A -85,B 0,C 180,E1 16035.786,E2 16035.786} C_VEL
LIN {X 0,Y 367.663,Z 403.986,A -85,B 0,C 180,E1 16034.167,E2 16034.167} C_VEL
LIN {X 0,Y 365.469,Z 400.338,A -85,B 0,C 180,E1 16032.963,E2 16032.963} C_VEL
LIN {X 0,Y 362.208,Z 398.073,A -85,B 0,C 180,E1 16031.302,E2 16031.302} C_VEL
LIN {X 0,Y 360.115,Z 394.676,A -85,B 0,C 180,E1 16029.993,E2 16029.993} C_VEL
LIN {X 0,Y 359.24,Z 393.61,A -85,B 0,C 180,E1 16029.451,E2 16029.451} C_VEL
LIN {X 0,Y 355.902,Z 391.384,A -85,B 0,C 180,E1 16027.425,E2 16027.425} C_VEL
LIN {X 0,Y 354.17,Z 388.542,A -85,B 0,C 180,E1 16026.077,E2 16026.077} C_VEL
LIN {X 0,Y 353.864,Z 387.11,A -85,B 0,C 180,E1 16025.146,E2 16025.146} C_VEL
LIN {X 0,Y 353.848,Z 386.955,A -85,B 0,C 180,E1 16020.971,E2 16020.971} C_VEL
LIN {X 0,Y 353.848,Z 386.958,A -85,B 0,C 180,E1 16016.922,E2 16016.922} C_VEL
LIN {X 0,Y 353.852,Z 386.969,A -85,B 0,C 180,E1 16012.694,E2 16012.694} C_VEL
LIN {X 0,Y 353.853,Z 386.969,A -85,B 0,C 180,E1 16008.591,E2 16008.591} C_VEL
LIN {X 0,Y 353.855,Z 386.959,A -85,B 0,C 180,E1 16004.428,E2 16004.428} C_VEL
LIN {X 0,Y 353.848,Z 386.954,A -85,B 0,C 180,E1 16000.179,E2 16000.179} C_VEL
LIN {X 0,Y 353.856,Z 386.954,A -85,B 0,C 180,E1 15996.167,E2 15996.167} C_VEL
LIN {X 0,Y 353.861,Z 386.957,A -85,B 0,C 180,E1 15992.027,E2 15992.027} C_VEL
LIN {X 0,Y 353.862,Z 386.966,A -85,B 0,C 180,E1 15987.913,E2 15987.913} C_VEL
LIN {X 0,Y 353.86,Z 386.964,A -85,B 0,C 180,E1 15983.804,E2 15983.804} C_VEL
LIN {X 0,Y 353.931,Z 387.377,A -85,B 0,C 180,E1 15981.744,E2 15981.744} C_VEL
LIN {X 0,Y 354.369,Z 388.998,A -85,B 0,C 180,E1 15980.956,E2 15980.956} C_VEL
LIN {X 0,Y 356.494,Z 391.96,A -85,B 0,C 180,E1 15979.406,E2 15979.406} C_VEL
LIN {X 0,Y 359.999,Z 394.263,A -85,B 0,C 180,E1 15977.336,E2 15977.336} C_VEL
LIN {X 0,Y 361.933,Z 397.722,A -85,B 0,C 180,E1 15976.099,E2 15976.099} C_VEL
LIN {X 0,Y 364.968,Z 400.091,A -85,B 0,C 180,E1 15974.526,E2 15974.526} C_VEL
LIN {X 0,Y 365.818,Z 400.737,A -85,B 0,C 180,E1 15974.103,E2 15974.103} C_VEL
LIN {X 0,Y 368,Z 404.326,A -85,B 0,C 180,E1 15972.925,E2 15972.925} C_VEL
LIN {X 0,Y 371.505,Z 407.324,A -85,B 0,C 180,E1 15971.332,E2 15971.332} C_VEL
LIN {X 0,Y 374.338,Z 411.332,A -85,B 0,C 180,E1 15970.026,E2 15970.026} C_VEL
LIN {X 0,Y 376.88,Z 413.643,A -85,B 0,C 180,E1 15968.983,E2 15968.983} C_VEL
LIN {X 0,Y 380.14,Z 417.875,A -85,B 0,C 180,E1 15967.655,E2 15967.655} C_VEL
LIN {X 0,Y 382.069,Z 419.827,A -85,B 0,C 180,E1 15966.919,E2 15966.919} C_VEL
LIN {X 0,Y 385.804,Z 424.379,A -85,B 0,C 180,E1 15965.533,E2 15965.533} C_VEL
LIN {X 0,Y 392.188,Z 432.167,A -85,B 0,C 180,E1 15963.33,E2 15963.33} C_VEL
LIN {X 0,Y 397.002,Z 438.282,A -85,B 0,C 180,E1 15961.787,E2 15961.787} C_VEL
LIN {X 0,Y 404.548,Z 447.858,A -85,B 0,C 180,E1 15959.543,E2 15959.543} C_VEL
LIN {X 0,Y 415.575,Z 462.843,A -85,B 0,C 180,E1 15956.558,E2 15956.558} C_VEL
LIN {X 0,Y 425.425,Z 477.15,A -85,B 0,C 180,E1 15954.139,E2 15954.139} C_VEL
LIN {X 0,Y 414.485,Z 684.736,A -85,B 0,C 180,E1 15950.108,E2 15950.108} C_VEL
LIN {X 0,Y 412.389,Z 719.839,A -85,B 0,C 180,E1 15949.385,E2 15949.385} C_VEL
LIN {X 0,Y 410.062,Z 741.901,A -85,B 0,C 180,E1 15948.738,E2 15948.738} C_VEL
LIN {X 0,Y 406.752,Z 765.884,A -85,B 0,C 180,E1 15947.779,E2 15947.779} C_VEL
LIN {X 0,Y 403.212,Z 786.7,A -85,B 0,C 180,E1 15946.713,E2 15946.713} C_VEL
LIN {X 0,Y 398.839,Z 808.325,A -85,B 0,C 180,E1 15945.332,E2 15945.332} C_VEL
LIN {X 0,Y 398.216,Z 811.184,A -85,B 0,C 180,E1 15945.129,E2 15945.129} C_VEL
LIN {X 0,Y 395.988,Z 818.108,A -85,B 0,C 180,E1 15944.726,E2 15944.726} C_VEL
LIN {X 0,Y 387.492,Z 835.484,A -85,B 0,C 180,E1 15943.922,E2 15943.922} C_VEL
LIN {X 0,Y 385.024,Z 841.963,A -85,B 0,C 180,E1 15943.411,E2 15943.411} C_VEL
LIN {X 0,Y 379.81,Z 860.443,A -85,B 0,C 180,E1 15941.46,E2 15941.46} C_VEL
LIN {X 0,Y 374.326,Z 878.852,A -85,B 0,C 180,E1 15939.177,E2 15939.177} C_VEL
LIN {X 0,Y 369.293,Z 894.761,A -85,B 0,C 180,E1 15936.838,E2 15936.838} C_VEL
LIN {X 0,Y 363.776,Z 911.913,A -85,B 0,C 180,E1 15933.86,E2 15933.86} C_VEL
LIN {X 0,Y 359.188,Z 926.106,A -85,B 0,C 180,E1 15930.953,E2 15930.953} C_VEL
LIN {X 0,Y 354.989,Z 939.301,A -85,B 0,C 180,E1 15927.736,E2 15927.736} C_VEL
LIN {X 0,Y 351.572,Z 950.805,A -85,B 0,C 180,E1 15924.447,E2 15924.447} C_VEL
LIN {X 0,Y 348.743,Z 960.968,A -85,B 0,C 180,E1 15920.923,E2 15920.923} C_VEL
LIN {X 0,Y 346.614,Z 969.988,A -85,B 0,C 180,E1 15917.163,E2 15917.163} C_VEL
LIN {X 0,Y 345.312,Z 976.655,A -85,B 0,C 180,E1 15913.684,E2 15913.684} C_VEL
LIN {X 0,Y 344.456,Z 982.509,A -85,B 0,C 180,E1 15909.788,E2 15909.788} C_VEL
LIN {X 0,Y 344.103,Z 986.054,A -85,B 0,C 180,E1 15906.538,E2 15906.538} C_VEL
LIN {X 0,Y 343.968,Z 988.703,A -85,B 0,C 180,E1 15903.03,E2 15903.03} C_VEL
LIN {X 0,Y 343.93,Z 989.893,A -85,B 0,C 180,E1 15899.609,E2 15899.609} C_VEL
LIN {X 0,Y 343.932,Z 989.938,A -85,B 0,C 180,E1 15896.467,E2 15896.467} C_VEL
LIN {X 0,Y 343.968,Z 988.853,A -85,B 0,C 180,E1 15893.003,E2 15893.003} C_VEL
LIN {X 0,Y 344.103,Z 986.378,A -85,B 0,C 180,E1 15889.579,E2 15889.579} C_VEL
LIN {X 0,Y 344.445,Z 982.894,A -85,B 0,C 180,E1 15886.287,E2 15886.287} C_VEL
LIN {X 0,Y 345.292,Z 977.226,A -85,B 0,C 180,E1 15882.4,E2 15882.4} C_VEL
LIN {X 0,Y 346.556,Z 970.8,A -85,B 0,C 180,E1 15878.974,E2 15878.974} C_VEL
LIN {X 0,Y 348.68,Z 961.957,A -85,B 0,C 180,E1 15875.185,E2 15875.185} C_VEL
LIN {X 0,Y 351.445,Z 952.158,A -85,B 0,C 180,E1 15871.712,E2 15871.712} C_VEL
LIN {X 0,Y 354.97,Z 940.567,A -85,B 0,C 180,E1 15868.311,E2 15868.311} C_VEL
LIN {X 0,Y 359.297,Z 927.38,A -85,B 0,C 180,E1 15865.024,E2 15865.024} C_VEL
LIN {X 0,Y 363.932,Z 913.41,A -85,B 0,C 180,E1 15862.111,E2 15862.111} C_VEL
LIN {X 0,Y 369.456,Z 896.867,A -85,B 0,C 180,E1 15859.172,E2 15859.172} C_VEL
LIN {X 0,Y 374.8,Z 880.484,A -85,B 0,C 180,E1 15856.716,E2 15856.716} C_VEL
LIN {X 0,Y 380.33,Z 862.719,A -85,B 0,C 180,E1 15854.463,E2 15854.463} C_VEL
LIN {X 0,Y 385.674,Z 844.529,A -85,B 0,C 180,E1 15852.502,E2 15852.502} C_VEL
LIN {X 0,Y 391.024,Z 824.391,A -85,B 0,C 180,E1 15850.691,E2 15850.691} C_VEL
LIN {X 0,Y 395.994,Z 803.807,A -85,B 0,C 180,E1 15849.148,E2 15849.148} C_VEL
LIN {X 0,Y 400.375,Z 782.607,A -85,B 0,C 180,E1 15847.859,E2 15847.859} C_VEL
LIN {X 0,Y 404.539,Z 758.695,A -85,B 0,C 180,E1 15846.707,E2 15846.707} C_VEL
LIN {X 0,Y 407.641,Z 736.322,A -85,B 0,C 180,E1 15845.884,E2 15845.884} C_VEL
LIN {X 0,Y 409.904,Z 713.209,A -85,B 0,C 180,E1 15845.277,E2 15845.277} C_VEL
LIN {X 0,Y 423.21,Z 508.568,A -85,B 0,C 180,E1 15841.122,E2 15841.122} C_VEL
LIN {X 0,Y 424.972,Z 482.604,A -85,B 0,C 180,E1 15840.572,E2 15840.572} C_VEL
LIN {X 0,Y 418.296,Z 471.691,A -85,B 0,C 180,E1 15838.281,E2 15838.281} C_VEL
LIN {X 0,Y 412.697,Z 463.077,A -85,B 0,C 180,E1 15836.01,E2 15836.01} C_VEL
LIN {X 0,Y 409.316,Z 458.154,A -85,B 0,C 180,E1 15834.393,E2 15834.393} C_VEL
LIN {X 0,Y 406.279,Z 453.67,A -85,B 0,C 180,E1 15832.665,E2 15832.665} C_VEL
LIN {X 0,Y 403.35,Z 449.122,A -85,B 0,C 180,E1 15830.519,E2 15830.519} C_VEL
LIN {X 0,Y 400.367,Z 445.276,A -85,B 0,C 180,E1 15827.085,E2 15827.085} C_VEL
LIN {X 0,Y 399.908,Z 443.668,A -85,B 0,C 180,E1 15825.67,E2 15825.67} C_VEL
LIN {X 0,Y 399.919,Z 443.692,A -85,B 0,C 180,E1 15822.692,E2 15822.692} C_VEL
LIN {X 0,Y 402.224,Z 448.156,A -85,B 0,C 180,E1 15818.873,E2 15818.873} C_VEL
LIN {X 0,Y 403.467,Z 449.46,A -85,B 0,C 180,E1 15817.796,E2 15817.796} C_VEL
LIN {X 0,Y 406.354,Z 453.729,A -85,B 0,C 180,E1 15815.738,E2 15815.738} C_VEL
LIN {X 0,Y 409.897,Z 459.431,A -85,B 0,C 180,E1 15813.722,E2 15813.722} C_VEL
LIN {X 0,Y 414.334,Z 466.913,A -85,B 0,C 180,E1 15811.655,E2 15811.655} C_VEL
LIN {X 0,Y 420.053,Z 477.108,A -85,B 0,C 180,E1 15809.417,E2 15809.417} C_VEL
LIN {X 0,Y 424.944,Z 486.511,A -85,B 0,C 180,E1 15807.734,E2 15807.734} C_VEL
LIN {X 0,Y 412.897,Z 669.595,A -85,B 0,C 180,E1 15804.012,E2 15804.012} C_VEL
LIN {X 0,Y 408.718,Z 736.115,A -85,B 0,C 180,E1 15802.645,E2 15802.645} C_VEL
LIN {X 0,Y 405.961,Z 759.233,A -85,B 0,C 180,E1 15801.992,E2 15801.992} C_VEL
LIN {X 0,Y 402.516,Z 781.727,A -85,B 0,C 180,E1 15801.149,E2 15801.149} C_VEL
LIN {X 0,Y 398.619,Z 802.471,A -85,B 0,C 180,E1 15800.137,E2 15800.137} C_VEL
LIN {X 0,Y 393.924,Z 824.278,A -85,B 0,C 180,E1 15798.818,E2 15798.818} C_VEL
LIN {X 0,Y 388.997,Z 844.465,A -85,B 0,C 180,E1 15797.321,E2 15797.321} C_VEL
LIN {X 0,Y 383.298,Z 865.754,A -85,B 0,C 180,E1 15795.413,E2 15795.413} C_VEL
LIN {X 0,Y 377.914,Z 884.634,A -85,B 0,C 180,E1 15793.393,E2 15793.393} C_VEL
LIN {X 0,Y 372.493,Z 902.497,A -85,B 0,C 180,E1 15791.123,E2 15791.123} C_VEL
LIN {X 0,Y 367.183,Z 919.687,A -85,B 0,C 180,E1 15788.582,E2 15788.582} C_VEL
LIN {X 0,Y 362.053,Z 935.953,A -85,B 0,C 180,E1 15785.717,E2 15785.717} C_VEL
LIN {X 0,Y 357.478,Z 950.859,A -85,B 0,C 180,E1 15782.661,E2 15782.661} C_VEL
LIN {X 0,Y 353.561,Z 964.172,A -85,B 0,C 180,E1 15779.425,E2 15779.425} C_VEL
LIN {X 0,Y 350.082,Z 976.993,A -85,B 0,C 180,E1 15775.733,E2 15775.733} C_VEL
LIN {X 0,Y 347.603,Z 987.464,A -85,B 0,C 180,E1 15772.14,E2 15772.14} C_VEL
LIN {X 0,Y 345.867,Z 996.051,A -85,B 0,C 180,E1 15768.523,E2 15768.523} C_VEL
LIN {X 0,Y 344.796,Z 1003.025,A -85,B 0,C 180,E1 15764.961,E2 15764.961} C_VEL
LIN {X 0,Y 344.219,Z 1008.357,A -85,B 0,C 180,E1 15761.396,E2 15761.396} C_VEL
LIN {X 0,Y 344.006,Z 1012.134,A -85,B 0,C 180,E1 15758.024,E2 15758.024} C_VEL
LIN {X 0,Y 343.937,Z 1014.753,A -85,B 0,C 180,E1 15754.339,E2 15754.339} C_VEL
LIN {X 0,Y 343.936,Z 1015.75,A -85,B 0,C 180,E1 15751.17,E2 15751.17} C_VEL
LIN {X 0,Y 343.943,Z 1015.632,A -85,B 0,C 180,E1 15747.839,E2 15747.839} C_VEL
LIN {X 0,Y 343.942,Z 1013.939,A -85,B 0,C 180,E1 15744.165,E2 15744.165} C_VEL
LIN {X 0,Y 344.056,Z 1011.101,A -85,B 0,C 180,E1 15740.807,E2 15740.807} C_VEL
LIN {X 0,Y 344.457,Z 1006.196,A -85,B 0,C 180,E1 15736.919,E2 15736.919} C_VEL
LIN {X 0,Y 345.227,Z 1000.367,A -85,B 0,C 180,E1 15733.464,E2 15733.464} C_VEL
LIN {X 0,Y 346.706,Z 992.075,A -85,B 0,C 180,E1 15729.582,E2 15729.582} C_VEL
LIN {X 0,Y 348.707,Z 983.138,A -85,B 0,C 180,E1 15726.159,E2 15726.159} C_VEL
LIN {X 0,Y 351.656,Z 971.637,A -85,B 0,C 180,E1 15722.51,E2 15722.51} C_VEL
LIN {X 0,Y 355.276,Z 959.06,A -85,B 0,C 180,E1 15719.133,E2 15719.133} C_VEL
LIN {X 0,Y 359.503,Z 944.968,A -85,B 0,C 180,E1 15715.975,E2 15715.975} C_VEL
LIN {X 0,Y 364.532,Z 928.808,A -85,B 0,C 180,E1 15712.891,E2 15712.891} C_VEL
LIN {X 0,Y 369.386,Z 913.211,A -85,B 0,C 180,E1 15710.362,E2 15710.362} C_VEL
LIN {X 0,Y 375.016,Z 894.534,A -85,B 0,C 180,E1 15707.795,E2 15707.795} C_VEL
LIN {X 0,Y 380.486,Z 875.842,A -85,B 0,C 180,E1 15705.624,E2 15705.624} C_VEL
LIN {X 0,Y 385.599,Z 856.775,A -85,B 0,C 180,E1 15703.776,E2 15703.776} C_VEL
LIN {X 0,Y 390.706,Z 836.383,A -85,B 0,C 180,E1 15702.104,E2 15702.104} C_VEL
LIN {X 0,Y 395.256,Z 815.624,A -85,B 0,C 180,E1 15700.714,E2 15700.714} C_VEL
LIN {X 0,Y 399.606,Z 792.962,A -85,B 0,C 180,E1 15699.483,E2 15699.483} C_VEL
LIN {X 0,Y 403.048,Z 771.336,A -85,B 0,C 180,E1 15698.567,E2 15698.567} C_VEL
LIN {X 0,Y 406.081,Z 747.116,A -85,B 0,C 180,E1 15697.807,E2 15697.807} C_VEL
LIN {X 0,Y 407.999,Z 723.432,A -85,B 0,C 180,E1 15697.261,E2 15697.261} C_VEL
LIN {X 0,Y 419.188,Z 516.362,A -85,B 0,C 180,E1 15693.209,E2 15693.209} C_VEL
LIN {X 0,Y 420.858,Z 485.765,A -85,B 0,C 180,E1 15692.595,E2 15692.595} C_VEL
LIN {X 0,Y 409.828,Z 468.428,A -85,B 0,C 180,E1 15689.727,E2 15689.727} C_VEL
LIN {X 0,Y 400.001,Z 453.954,A -85,B 0,C 180,E1 15686.899,E2 15686.899} C_VEL
LIN {X 0,Y 392.999,Z 444.299,A -85,B 0,C 180,E1 15684.7,E2 15684.7} C_VEL
LIN {X 0,Y 386.898,Z 436.013,A -85,B 0,C 180,E1 15682.607,E2 15682.607} C_VEL
LIN {X 0,Y 382.988,Z 431.163,A -85,B 0,C 180,E1 15681.197,E2 15681.197} C_VEL
LIN {X 0,Y 378.815,Z 426.006,A -85,B 0,C 180,E1 15679.585,E2 15679.585} C_VEL
LIN {X 0,Y 375.137,Z 421.696,A -85,B 0,C 180,E1 15678.089,E2 15678.089} C_VEL
LIN {X 0,Y 373.965,Z 420.22,A -85,B 0,C 180,E1 15677.585,E2 15677.585} C_VEL
LIN {X 0,Y 370.498,Z 416.485,A -85,B 0,C 180,E1 15676.058,E2 15676.058} C_VEL
LIN {X 0,Y 368.962,Z 414.233,A -85,B 0,C 180,E1 15675.32,E2 15675.32} C_VEL
LIN {X 0,Y 365.538,Z 411.107,A -85,B 0,C 180,E1 15673.686,E2 15673.686} C_VEL
LIN {X 0,Y 363.775,Z 408.052,A -85,B 0,C 180,E1 15672.702,E2 15672.702} C_VEL
LIN {X 0,Y 360.431,Z 405.563,A -85,B 0,C 180,E1 15670.954,E2 15670.954} C_VEL
LIN {X 0,Y 358.244,Z 401.994,A -85,B 0,C 180,E1 15669.559,E2 15669.559} C_VEL
LIN {X 0,Y 357.323,Z 401.218,A -85,B 0,C 180,E1 15669.015,E2 15669.015} C_VEL
LIN {X 0,Y 354.226,Z 398.886,A -85,B 0,C 180,E1 15667.052,E2 15667.052} C_VEL
LIN {X 0,Y 352.406,Z 395.924,A -85,B 0,C 180,E1 15665.658,E2 15665.658} C_VEL
LIN {X 0,Y 351.418,Z 394.646,A -85,B 0,C 180,E1 15664.896,E2 15664.896} C_VEL
LIN {X 0,Y 347.876,Z 392.328,A -85,B 0,C 180,E1 15662.058,E2 15662.058} C_VEL
LIN {X 0,Y 345.983,Z 388.566,A -85,B 0,C 180,E1 15659.668,E2 15659.668} C_VEL
LIN {X 0,Y 345.878,Z 387.962,A -85,B 0,C 180,E1 15657.846,E2 15657.846} C_VEL
LIN {X 0,Y 345.883,Z 387.947,A -85,B 0,C 180,E1 15653.693,E2 15653.693} C_VEL
LIN {X 0,Y 345.887,Z 387.954,A -85,B 0,C 180,E1 15649.507,E2 15649.507} C_VEL
LIN {X 0,Y 345.89,Z 387.962,A -85,B 0,C 180,E1 15645.434,E2 15645.434} C_VEL
LIN {X 0,Y 345.895,Z 387.957,A -85,B 0,C 180,E1 15641.284,E2 15641.284} C_VEL
LIN {X 0,Y 345.893,Z 387.95,A -85,B 0,C 180,E1 15637.21,E2 15637.21} C_VEL
LIN {X 0,Y 345.899,Z 387.944,A -85,B 0,C 180,E1 15633.01,E2 15633.01} C_VEL
LIN {X 0,Y 345.912,Z 387.992,A -85,B 0,C 180,E1 15628.813,E2 15628.813} C_VEL
LIN {X 0,Y 346.05,Z 388.796,A -85,B 0,C 180,E1 15627.295,E2 15627.295} C_VEL
LIN {X 0,Y 348.118,Z 392.555,A -85,B 0,C 180,E1 15624.932,E2 15624.932} C_VEL
LIN {X 0,Y 352.171,Z 395.328,A -85,B 0,C 180,E1 15621.761,E2 15621.761} C_VEL
LIN {X 0,Y 354.005,Z 398.597,A -85,B 0,C 180,E1 15620.333,E2 15620.333} C_VEL
LIN {X 0,Y 357.025,Z 401.051,A -85,B 0,C 180,E1 15618.386,E2 15618.386} C_VEL
LIN {X 0,Y 358.225,Z 401.869,A -85,B 0,C 180,E1 15617.693,E2 15617.693} C_VEL
LIN {X 0,Y 360.407,Z 405.499,A -85,B 0,C 180,E1 15616.307,E2 15616.307} C_VEL
LIN {X 0,Y 363.996,Z 408.456,A -85,B 0,C 180,E1 15614.422,E2 15614.422} C_VEL
LIN {X 0,Y 366.6,Z 412.305,A -85,B 0,C 180,E1 15613.034,E2 15613.034} C_VEL
LIN {X 0,Y 369.522,Z 414.836,A -85,B 0,C 180,E1 15611.685,E2 15611.685} C_VEL
LIN {X 0,Y 372.652,Z 419.053,A -85,B 0,C 180,E1 15610.24,E2 15610.24} C_VEL
LIN {X 0,Y 374.831,Z 421.147,A -85,B 0,C 180,E1 15609.324,E2 15609.324} C_VEL
LIN {X 0,Y 378.27,Z 425.48,A -85,B 0,C 180,E1 15607.907,E2 15607.907} C_VEL
LIN {X 0,Y 380.004,Z 427.381,A -85,B 0,C 180,E1 15607.235,E2 15607.235} C_VEL
LIN {X 0,Y 384.004,Z 432.087,A -85,B 0,C 180,E1 15605.734,E2 15605.734} C_VEL
LIN {X 0,Y 388.604,Z 437.722,A -85,B 0,C 180,E1 15604.112,E2 15604.112} C_VEL
LIN {X 0,Y 398.166,Z 450.11,A -85,B 0,C 180,E1 15601.025,E2 15601.025} C_VEL
LIN {X 0,Y 405.991,Z 460.573,A -85,B 0,C 180,E1 15598.747,E2 15598.747} C_VEL
LIN {X 0,Y 415.451,Z 473.78,A -85,B 0,C 180,E1 15596.229,E2 15596.229} C_VEL
LIN {X 0,Y 420.583,Z 481.38,A -85,B 0,C 180,E1 15594.948,E2 15594.948} C_VEL
LIN {X 0,Y 409.184,Z 689.104,A -85,B 0,C 180,E1 15590.887,E2 15590.887} C_VEL
LIN {X 0,Y 407.062,Z 721.656,A -85,B 0,C 180,E1 15590.198,E2 15590.198} C_VEL
LIN {X 0,Y 404.652,Z 743.589,A -85,B 0,C 180,E1 15589.542,E2 15589.542} C_VEL
LIN {X 0,Y 401.387,Z 766.211,A -85,B 0,C 180,E1 15588.626,E2 15588.626} C_VEL
LIN {X 0,Y 397.724,Z 787.074,A -85,B 0,C 180,E1 15587.554,E2 15587.554} C_VEL
LIN {X 0,Y 393.399,Z 807.774,A -85,B 0,C 180,E1 15586.23,E2 15586.23} C_VEL
LIN {X 0,Y 388.85,Z 827.13,A -85,B 0,C 180,E1 15584.743,E2 15584.743} C_VEL
LIN {X 0,Y 385.024,Z 841.963,A -85,B 0,C 180,E1 15583.411,E2 15583.411} C_VEL
LIN {X 0,Y 382.5,Z 848.392,A -85,B 0,C 180,E1 15582.869,E2 15582.869} C_VEL
LIN {X 0,Y 373.311,Z 864.659,A -85,B 0,C 180,E1 15581.731,E2 15581.731} C_VEL
LIN {X 0,Y 370.695,Z 870.632,A -85,B 0,C 180,E1 15581.097,E2 15581.097} C_VEL
LIN {X 0,Y 365.054,Z 888.415,A -85,B 0,C 180,E1 15578.66,E2 15578.66} C_VEL
LIN {X 0,Y 359.688,Z 904.309,A -85,B 0,C 180,E1 15576.059,E2 15576.059} C_VEL
LIN {X 0,Y 354.475,Z 919.694,A -85,B 0,C 180,E1 15573.112,E2 15573.112} C_VEL
LIN {X 0,Y 349.953,Z 933.004,A -85,B 0,C 180,E1 15570.08,E2 15570.08} C_VEL
LIN {X 0,Y 345.606,Z 946.334,A -85,B 0,C 180,E1 15566.478,E2 15566.478} C_VEL
LIN {X 0,Y 342.428,Z 956.784,A -85,B 0,C 180,E1 15563.109,E2 15563.109} C_VEL
LIN {X 0,Y 339.765,Z 966.467,A -85,B 0,C 180,E1 15559.312,E2 15559.312} C_VEL
LIN {X 0,Y 337.996,Z 974.253,A -85,B 0,C 180,E1 15555.608,E2 15555.608} C_VEL
LIN {X 0,Y 336.849,Z 980.388,A -85,B 0,C 180,E1 15551.836,E2 15551.836} C_VEL
LIN {X 0,Y 336.277,Z 985.013,A -85,B 0,C 180,E1 15548.178,E2 15548.178} C_VEL
LIN {X 0,Y 336.014,Z 988.154,A -85,B 0,C 180,E1 15544.435,E2 15544.435} C_VEL
LIN {X 0,Y 335.972,Z 989.883,A -85,B 0,C 180,E1 15540.978,E2 15540.978} C_VEL
LIN {X 0,Y 335.944,Z 990.332,A -85,B 0,C 180,E1 15537.198,E2 15537.198} C_VEL
LIN {X 0,Y 335.96,Z 989.541,A -85,B 0,C 180,E1 15533.891,E2 15533.891} C_VEL
LIN {X 0,Y 336.111,Z 987.254,A -85,B 0,C 180,E1 15530.013,E2 15530.013} C_VEL
LIN {X 0,Y 336.449,Z 983.671,A -85,B 0,C 180,E1 15526.409,E2 15526.409} C_VEL
LIN {X 0,Y 337.292,Z 978.382,A -85,B 0,C 180,E1 15522.523,E2 15522.523} C_VEL
LIN {X 0,Y 338.59,Z 972.015,A -85,B 0,C 180,E1 15518.976,E2 15518.976} C_VEL
LIN {X 0,Y 340.785,Z 963.462,A -85,B 0,C 180,E1 15515.105,E2 15515.105} C_VEL
LIN {X 0,Y 343.588,Z 953.906,A -85,B 0,C 180,E1 15511.589,E2 15511.589} C_VEL
LIN {X 0,Y 347.448,Z 941.997,A -85,B 0,C 180,E1 15507.932,E2 15507.932} C_VEL
LIN {X 0,Y 351.783,Z 929.448,A -85,B 0,C 180,E1 15504.697,E2 15504.697} C_VEL
LIN {X 0,Y 356.751,Z 915.292,A -85,B 0,C 180,E1 15501.632,E2 15501.632} C_VEL
LIN {X 0,Y 362.241,Z 899.823,A -85,B 0,C 180,E1 15498.775,E2 15498.775} C_VEL
LIN {X 0,Y 367.975,Z 882.989,A -85,B 0,C 180,E1 15496.172,E2 15496.172} C_VEL
LIN {X 0,Y 374.304,Z 863.725,A -85,B 0,C 180,E1 15493.667,E2 15493.667} C_VEL
LIN {X 0,Y 379.623,Z 846.424,A -85,B 0,C 180,E1 15491.771,E2 15491.771} C_VEL
LIN {X 0,Y 385.458,Z 825.56,A -85,B 0,C 180,E1 15489.858,E2 15489.858} C_VEL
LIN {X 0,Y 390.6,Z 805.322,A -85,B 0,C 180,E1 15488.316,E2 15488.316} C_VEL
LIN {X 0,Y 395.309,Z 783.474,A -85,B 0,C 180,E1 15486.974,E2 15486.974} C_VEL
LIN {X 0,Y 399.567,Z 760.287,A -85,B 0,C 180,E1 15485.84,E2 15485.84} C_VEL
LIN {X 0,Y 402.709,Z 738.629,A -85,B 0,C 180,E1 15485.027,E2 15485.027} C_VEL
LIN {X 0,Y 405.258,Z 714.517,A -85,B 0,C 180,E1 15484.376,E2 15484.376} C_VEL
LIN {X 0,Y 419.4,Z 508.806,A -85,B 0,C 180,E1 15480.163,E2 15480.163} C_VEL
LIN {X 0,Y 420.957,Z 487.161,A -85,B 0,C 180,E1 15479.703,E2 15479.703} C_VEL
LIN {X 0,Y 414.808,Z 477.044,A -85,B 0,C 180,E1 15477.445,E2 15477.445} C_VEL
LIN {X 0,Y 410.154,Z 469.705,A -85,B 0,C 180,E1 15475.424,E2 15475.424} C_VEL
LIN {X 0,Y 407.37,Z 465.46,A -85,B 0,C 180,E1 15474.013,E2 15474.013} C_VEL
LIN {X 0,Y 404.583,Z 461.176,A -85,B 0,C 180,E1 15472.331,E2 15472.331} C_VEL
LIN {X 0,Y 401.722,Z 456.63,A -85,B 0,C 180,E1 15470.112,E2 15470.112} C_VEL
LIN {X 0,Y 399.152,Z 453.076,A -85,B 0,C 180,E1 15466.898,E2 15466.898} C_VEL
LIN {X 0,Y 398.783,Z 451.584,A -85,B 0,C 180,E1 15465.628,E2 15465.628} C_VEL
LIN {X 0,Y 398.819,Z 451.659,A -85,B 0,C 180,E1 15462.643,E2 15462.643} C_VEL
LIN {X 0,Y 400.722,Z 455.753,A -85,B 0,C 180,E1 15459.249,E2 15459.249} C_VEL
LIN {X 0,Y 402.052,Z 457.221,A -85,B 0,C 180,E1 15458.021,E2 15458.021} C_VEL
LIN {X 0,Y 405.489,Z 462.535,A -85,B 0,C 180,E1 15455.528,E2 15455.528} C_VEL
LIN {X 0,Y 409.227,Z 468.815,A -85,B 0,C 180,E1 15453.441,E2 15453.441} C_VEL
LIN {X 0,Y 413.963,Z 477.435,A -85,B 0,C 180,E1 15451.258,E2 15451.258} C_VEL
LIN {X 0,Y 420.004,Z 488.774,A -85,B 0,C 180,E1 15448.937,E2 15448.937} C_VEL
LIN {X 0,Y 420.9,Z 490.959,A -85,B 0,C 180,E1 15448.608,E2 15448.608} C_VEL
LIN {X 0,Y 408.327,Z 672.397,A -85,B 0,C 180,E1 15444.893,E2 15444.893} C_VEL
LIN {X 0,Y 404.088,Z 735.846,A -85,B 0,C 180,E1 15443.574,E2 15443.574} C_VEL
LIN {X 0,Y 401.204,Z 759.155,A -85,B 0,C 180,E1 15442.914,E2 15442.914} C_VEL
LIN {X 0,Y 397.531,Z 782.022,A -85,B 0,C 180,E1 15442.05,E2 15442.05} C_VEL
LIN {X 0,Y 393.758,Z 801.312,A -85,B 0,C 180,E1 15441.107,E2 15441.107} C_VEL
LIN {X 0,Y 388.882,Z 823.255,A -85,B 0,C 180,E1 15439.788,E2 15439.788} C_VEL
LIN {X 0,Y 383.742,Z 843.443,A -85,B 0,C 180,E1 15438.291,E2 15438.291} C_VEL
LIN {X 0,Y 377.559,Z 865.561,A -85,B 0,C 180,E1 15436.303,E2 15436.303} C_VEL
LIN {X 0,Y 371.869,Z 884.579,A -85,B 0,C 180,E1 15434.249,E2 15434.249} C_VEL
LIN {X 0,Y 366.019,Z 902.945,A -85,B 0,C 180,E1 15431.879,E2 15431.879} C_VEL
LIN {X 0,Y 360.44,Z 920.092,A -85,B 0,C 180,E1 15429.291,E2 15429.291} C_VEL
LIN {X 0,Y 355.163,Z 935.945,A -85,B 0,C 180,E1 15426.446,E2 15426.446} C_VEL
LIN {X 0,Y 350.171,Z 951.3,A -85,B 0,C 180,E1 15423.217,E2 15423.217} C_VEL
LIN {X 0,Y 346.137,Z 964.284,A -85,B 0,C 180,E1 15419.986,E2 15419.986} C_VEL
LIN {X 0,Y 342.556,Z 976.644,A -85,B 0,C 180,E1 15416.342,E2 15416.342} C_VEL
LIN {X 0,Y 339.9,Z 987.122,A -85,B 0,C 180,E1 15412.67,E2 15412.67} C_VEL
LIN {X 0,Y 338.051,Z 995.668,A -85,B 0,C 180,E1 15408.991,E2 15408.991} C_VEL
LIN {X 0,Y 336.871,Z 1002.759,A -85,B 0,C 180,E1 15405.288,E2 15405.288} C_VEL
LIN {X 0,Y 336.247,Z 1008.037,A -85,B 0,C 180,E1 15401.67,E2 15401.67} C_VEL
LIN {X 0,Y 336.021,Z 1011.821,A -85,B 0,C 180,E1 15398.216,E2 15398.216} C_VEL
LIN {X 0,Y 335.941,Z 1014.463,A -85,B 0,C 180,E1 15394.404,E2 15394.404} C_VEL
LIN {X 0,Y 335.943,Z 1015.449,A -85,B 0,C 180,E1 15391.198,E2 15391.198} C_VEL
LIN {X 0,Y 335.948,Z 1015.356,A -85,B 0,C 180,E1 15387.958,E2 15387.958} C_VEL
LIN {X 0,Y 335.944,Z 1013.755,A -85,B 0,C 180,E1 15384.197,E2 15384.197} C_VEL
LIN {X 0,Y 336.058,Z 1010.963,A -85,B 0,C 180,E1 15380.759,E2 15380.759} C_VEL
LIN {X 0,Y 336.477,Z 1006.148,A -85,B 0,C 180,E1 15376.778,E2 15376.778} C_VEL
LIN {X 0,Y 337.288,Z 1000.345,A -85,B 0,C 180,E1 15373.234,E2 15373.234} C_VEL
LIN {X 0,Y 338.847,Z 992.149,A -85,B 0,C 180,E1 15369.268,E2 15369.268} C_VEL
LIN {X 0,Y 340.94,Z 983.319,A -85,B 0,C 180,E1 15365.789,E2 15365.789} C_VEL
LIN {X 0,Y 344.043,Z 971.933,A -85,B 0,C 180,E1 15362.064,E2 15362.064} C_VEL
LIN {X 0,Y 347.84,Z 959.41,A -85,B 0,C 180,E1 15358.617,E2 15358.617} C_VEL
LIN {X 0,Y 352.264,Z 945.412,A -85,B 0,C 180,E1 15355.398,E2 15355.398} C_VEL
LIN {X 0,Y 357.364,Z 929.902,A -85,B 0,C 180,E1 15352.353,E2 15352.353} C_VEL
LIN {X 0,Y 362.371,Z 914.458,A -85,B 0,C 180,E1 15349.792,E2 15349.792} C_VEL
LIN {X 0,Y 368.099,Z 896.425,A -85,B 0,C 180,E1 15347.237,E2 15347.237} C_VEL
LIN {X 0,Y 373.652,Z 878.179,A -85,B 0,C 180,E1 15345.062,E2 15345.062} C_VEL
LIN {X 0,Y 379.366,Z 858.026,A -85,B 0,C 180,E1 15343.048,E2 15343.048} C_VEL
LIN {X 0,Y 384.274,Z 839.247,A -85,B 0,C 180,E1 15341.473,E2 15341.473} C_VEL
LIN {X 0,Y 389.098,Z 818.486,A -85,B 0,C 180,E1 15340.033,E2 15340.033} C_VEL
LIN {X 0,Y 393.285,Z 798.141,A -85,B 0,C 180,E1 15338.875,E2 15338.875} C_VEL
LIN {X 0,Y 397.2,Z 775.227,A -85,B 0,C 180,E1 15337.849,E2 15337.849} C_VEL
LIN {X 0,Y 400.352,Z 752.788,A -85,B 0,C 180,E1 15337.083,E2 15337.083} C_VEL
LIN {X 0,Y 402.531,Z 729.13,A -85,B 0,C 180,E1 15336.505,E2 15336.505} C_VEL
LIN {X 0,Y 414.444,Z 518.535,A -85,B 0,C 180,E1 15332.349,E2 15332.349} C_VEL
LIN {X 0,Y 416.035,Z 489.845,A -85,B 0,C 180,E1 15331.757,E2 15331.757} C_VEL
LIN {X 0,Y 406.127,Z 474.123,A -85,B 0,C 180,E1 15329.093,E2 15329.093} C_VEL
LIN {X 0,Y 396.473,Z 459.719,A -85,B 0,C 180,E1 15326.228,E2 15326.228} C_VEL
LIN {X 0,Y 387.838,Z 447.623,A -85,B 0,C 180,E1 15323.391,E2 15323.391} C_VEL
LIN {X 0,Y 380.981,Z 438.675,A -85,B 0,C 180,E1 15320.911,E2 15320.911} C_VEL
LIN {X 0,Y 376.468,Z 433.185,A -85,B 0,C 180,E1 15319.147,E2 15319.147} C_VEL
LIN {X 0,Y 372.708,Z 428.52,A -85,B 0,C 180,E1 15317.565,E2 15317.565} C_VEL
LIN {X 0,Y 368.288,Z 423.563,A -85,B 0,C 180,E1 15315.591,E2 15315.591} C_VEL
LIN {X 0,Y 366.912,Z 421.674,A -85,B 0,C 180,E1 15314.922,E2 15314.922} C_VEL
LIN {X 0,Y 363.418,Z 418.214,A -85,B 0,C 180,E1 15313.2,E2 15313.2} C_VEL
LIN {X 0,Y 361.774,Z 415.6,A -85,B 0,C 180,E1 15312.287,E2 15312.287} C_VEL
LIN {X 0,Y 358.41,Z 412.737,A -85,B 0,C 180,E1 15310.447,E2 15310.447} C_VEL
LIN {X 0,Y 356.237,Z 409.187,A -85,B 0,C 180,E1 15309.042,E2 15309.042} C_VEL
LIN {X 0,Y 352.89,Z 406.78,A -85,B 0,C 180,E1 15306.916,E2 15306.916} C_VEL
LIN {X 0,Y 350.795,Z 403.527,A -85,B 0,C 180,E1 15305.315,E2 15305.315} C_VEL
LIN {X 0,Y 350.094,Z 402.499,A -85,B 0,C 180,E1 15304.75,E2 15304.75} C_VEL
LIN {X 0,Y 346.658,Z 400.27,A -85,B 0,C 180,E1 15301.983,E2 15301.983} C_VEL
LIN {X 0,Y 344.068,Z 396.015,A -85,B 0,C 180,E1 15299.167,E2 15299.167} C_VEL
LIN {X 0,Y 339.854,Z 393.208,A -85,B 0,C 180,E1 15293.75,E2 15293.75} C_VEL
LIN {X 0,Y 338.101,Z 389.689,A -85,B 0,C 180,E1 15288.571,E2 15288.571} C_VEL
LIN {X 0,Y 338.013,Z 389.136,A -85,B 0,C 180,E1 15284.56,E2 15284.56} C_VEL
LIN {X 0,Y 338.038,Z 389.342,A -85,B 0,C 180,E1 15280.294,E2 15280.294} C_VEL
LIN {X 0,Y 338.2,Z 390.161,A -85,B 0,C 180,E1 15277.58,E2 15277.58} C_VEL
LIN {X 0,Y 341.01,Z 394.284,A -85,B 0,C 180,E1 15271.641,E2 15271.641} C_VEL
LIN {X 0,Y 344.373,Z 396.297,A -85,B 0,C 180,E1 15267.708,E2 15267.708} C_VEL
LIN {X 0,Y 346.91,Z 400.492,A -85,B 0,C 180,E1 15265.001,E2 15265.001} C_VEL
LIN {X 0,Y 350.653,Z 403.102,A -85,B 0,C 180,E1 15262.033,E2 15262.033} C_VEL
LIN {X 0,Y 352.549,Z 406.349,A -85,B 0,C 180,E1 15260.558,E2 15260.558} C_VEL
LIN {X 0,Y 355.777,Z 408.95,A -85,B 0,C 180,E1 15258.452,E2 15258.452} C_VEL
LIN {X 0,Y 356.543,Z 409.621,A -85,B 0,C 180,E1 15257.991,E2 15257.991} C_VEL
LIN {X 0,Y 359.05,Z 413.452,A -85,B 0,C 180,E1 15256.42,E2 15256.42} C_VEL
LIN {X 0,Y 362.197,Z 416.132,A -85,B 0,C 180,E1 15254.736,E2 15254.736} C_VEL
LIN {X 0,Y 365.087,Z 420.138,A -85,B 0,C 180,E1 15253.202,E2 15253.202} C_VEL
LIN {X 0,Y 367.608,Z 422.422,A -85,B 0,C 180,E1 15252.012,E2 15252.012} C_VEL
LIN {X 0,Y 371.037,Z 426.839,A -85,B 0,C 180,E1 15250.423,E2 15250.423} C_VEL
LIN {X 0,Y 372.882,Z 428.765,A -85,B 0,C 180,E1 15249.63,E2 15249.63} C_VEL
LIN {X 0,Y 376.615,Z 433.277,A -85,B 0,C 180,E1 15248.078,E2 15248.078} C_VEL
LIN {X 0,Y 382.847,Z 440.972,A -85,B 0,C 180,E1 15245.686,E2 15245.686} C_VEL
LIN {X 0,Y 387.779,Z 447.131,A -85,B 0,C 180,E1 15243.947,E2 15243.947} C_VEL
LIN {X 0,Y 395.121,Z 456.549,A -85,B 0,C 180,E1 15241.56,E2 15241.56} C_VEL
LIN {X 0,Y 403.579,Z 468.04,A -85,B 0,C 180,E1 15239.045,E2 15239.045} C_VEL
LIN {X 0,Y 412.68,Z 480.962,A -85,B 0,C 180,E1 15236.576,E2 15236.576} C_VEL
LIN {X 0,Y 415.799,Z 485.835,A -85,B 0,C 180,E1 15235.769,E2 15235.769} C_VEL
LIN {X 0,Y 403.942,Z 693.637,A -85,B 0,C 180,E1 15231.683,E2 15231.683} C_VEL
LIN {X 0,Y 401.8,Z 723.64,A -85,B 0,C 180,E1 15231.027,E2 15231.027} C_VEL
LIN {X 0,Y 399.212,Z 746.156,A -85,B 0,C 180,E1 15230.335,E2 15230.335} C_VEL
LIN {X 0,Y 395.875,Z 767.833,A -85,B 0,C 180,E1 15229.432,E2 15229.432} C_VEL
LIN {X 0,Y 391.876,Z 789.678,A -85,B 0,C 180,E1 15228.286,E2 15228.286} C_VEL
LIN {X 0,Y 387.397,Z 809.967,A -85,B 0,C 180,E1 15226.952,E2 15226.952} C_VEL
LIN {X 0,Y 382.499,Z 829.952,A -85,B 0,C 180,E1 15225.381,E2 15225.381} C_VEL
LIN {X 0,Y 377.195,Z 849.055,A -85,B 0,C 180,E1 15223.563,E2 15223.563} C_VEL
LIN {X 0,Y 371.475,Z 868.196,A -85,B 0,C 180,E1 15221.406,E2 15221.406} C_VEL
LIN {X 0,Y 370.695,Z 870.632,A -85,B 0,C 180,E1 15221.097,E2 15221.097} C_VEL
LIN {X 0,Y 368.063,Z 876.697,A -85,B 0,C 180,E1 15220.429,E2 15220.429} C_VEL
LIN {X 0,Y 358.448,Z 891.544,A -85,B 0,C 180,E1 15218.927,E2 15218.927} C_VEL
LIN {X 0,Y 355.793,Z 896.961,A -85,B 0,C 180,E1 15218.165,E2 15218.165} C_VEL
LIN {X 0,Y 350.059,Z 913.168,A -85,B 0,C 180,E1 15215.24,E2 15215.24} C_VEL
LIN {X 0,Y 344.91,Z 927.697,A -85,B 0,C 180,E1 15212.155,E2 15212.155} C_VEL
LIN {X 0,Y 340.284,Z 940.744,A -85,B 0,C 180,E1 15208.817,E2 15208.817} C_VEL
LIN {X 0,Y 336.324,Z 952.623,A -85,B 0,C 180,E1 15205.221,E2 15205.221} C_VEL
LIN {X 0,Y 333.353,Z 962.217,A -85,B 0,C 180,E1 15201.718,E2 15201.718} C_VEL
LIN {X 0,Y 330.875,Z 971.445,A -85,B 0,C 180,E1 15197.607,E2 15197.607} C_VEL
LIN {X 0,Y 329.446,Z 978.001,A -85,B 0,C 180,E1 15193.963,E2 15193.963} C_VEL
LIN {X 0,Y 328.536,Z 983.408,A -85,B 0,C 180,E1 15190.067,E2 15190.067} C_VEL
LIN {X 0,Y 328.135,Z 986.889,A -85,B 0,C 180,E1 15186.66,E2 15186.66} C_VEL
LIN {X 0,Y 327.973,Z 989.509,A -85,B 0,C 180,E1 15182.784,E2 15182.784} C_VEL
LIN {X 0,Y 327.949,Z 990.528,A -85,B 0,C 180,E1 15179.388,E2 15179.388} C_VEL
LIN {X 0,Y 327.94,Z 990.507,A -85,B 0,C 180,E1 15176.082,E2 15176.082} C_VEL
LIN {X 0,Y 327.999,Z 989.131,A -85,B 0,C 180,E1 15172.209,E2 15172.209} C_VEL
LIN {X 0,Y 328.18,Z 986.691,A -85,B 0,C 180,E1 15168.811,E2 15168.811} C_VEL
LIN {X 0,Y 328.697,Z 982.848,A -85,B 0,C 180,E1 15165.108,E2 15165.108} C_VEL
LIN {X 0,Y 329.709,Z 977.193,A -85,B 0,C 180,E1 15161.225,E2 15161.225} C_VEL
LIN {X 0,Y 331.453,Z 970.047,A -85,B 0,C 180,E1 15157.326,E2 15157.326} C_VEL
LIN {X 0,Y 333.876,Z 961.494,A -85,B 0,C 180,E1 15153.636,E2 15153.636} C_VEL
LIN {X 0,Y 337.305,Z 951.028,A -85,B 0,C 180,E1 15149.868,E2 15149.868} C_VEL
LIN {X 0,Y 341.343,Z 939.51,A -85,B 0,C 180,E1 15146.439,E2 15146.439} C_VEL
LIN {X 0,Y 346.518,Z 925.435,A -85,B 0,C 180,E1 15142.926,E2 15142.926} C_VEL
LIN {X 0,Y 351.946,Z 910.962,A -85,B 0,C 180,E1 15139.882,E2 15139.882} C_VEL
LIN {X 0,Y 357.816,Z 894.909,A -85,B 0,C 180,E1 15137.062,E2 15137.062} C_VEL
LIN {X 0,Y 364.037,Z 877.542,A -85,B 0,C 180,E1 15134.474,E2 15134.474} C_VEL
LIN {X 0,Y 369.768,Z 860.445,A -85,B 0,C 180,E1 15132.335,E2 15132.335} C_VEL
LIN {X 0,Y 376.17,Z 840.049,A -85,B 0,C 180,E1 15130.189,E2 15130.189} C_VEL
LIN {X 0,Y 381.632,Z 820.877,A -85,B 0,C 180,E1 15128.513,E2 15128.513} C_VEL
LIN {X 0,Y 386.858,Z 800.195,A -85,B 0,C 180,E1 15127.02,E2 15127.02} C_VEL
LIN {X 0,Y 391.456,Z 779.425,A -85,B 0,C 180,E1 15125.791,E2 15125.791} C_VEL
LIN {X 0,Y 395.434,Z 757.522,A -85,B 0,C 180,E1 15124.769,E2 15124.769} C_VEL
LIN {X 0,Y 398.767,Z 734.982,A -85,B 0,C 180,E1 15123.954,E2 15123.954} C_VEL
LIN {X 0,Y 401.069,Z 712.239,A -85,B 0,C 180,E1 15123.368,E2 15123.368} C_VEL
LIN {X 0,Y 415.428,Z 513.393,A -85,B 0,C 180,E1 15119.272,E2 15119.272} C_VEL
LIN {X 0,Y 417.043,Z 491.818,A -85,B 0,C 180,E1 15118.804,E2 15118.804} C_VEL
LIN {X 0,Y 411.231,Z 481.859,A -85,B 0,C 180,E1 15116.481,E2 15116.481} C_VEL
LIN {X 0,Y 406.172,Z 473.665,A -85,B 0,C 180,E1 15114.01,E2 15114.01} C_VEL
LIN {X 0,Y 402.925,Z 468.706,A -85,B 0,C 180,E1 15112.013,E2 15112.013} C_VEL
LIN {X 0,Y 400.217,Z 464.301,A -85,B 0,C 180,E1 15109.783,E2 15109.783} C_VEL
LIN {X 0,Y 397.911,Z 460.771,A -85,B 0,C 180,E1 15106.634,E2 15106.634} C_VEL
LIN {X 0,Y 397.614,Z 459.469,A -85,B 0,C 180,E1 15105.436,E2 15105.436} C_VEL
LIN {X 0,Y 397.67,Z 459.548,A -85,B 0,C 180,E1 15102.742,E2 15102.742} C_VEL
LIN {X 0,Y 399.428,Z 463.553,A -85,B 0,C 180,E1 15099.429,E2 15099.429} C_VEL
LIN {X 0,Y 400.646,Z 464.976,A -85,B 0,C 180,E1 15098.248,E2 15098.248} C_VEL
LIN {X 0,Y 403.848,Z 470.136,A -85,B 0,C 180,E1 15095.811,E2 15095.811} C_VEL
LIN {X 0,Y 407.245,Z 476.137,A -85,B 0,C 180,E1 15093.813,E2 15093.813} C_VEL
LIN {X 0,Y 411.645,Z 484.444,A -85,B 0,C 180,E1 15091.69,E2 15091.69} C_VEL
LIN {X 0,Y 417.039,Z 495.004,A -85,B 0,C 180,E1 15089.511,E2 15089.511} C_VEL
LIN {X 0,Y 403.727,Z 677.687,A -85,B 0,C 180,E1 15085.746,E2 15085.746} C_VEL
LIN {X 0,Y 399.582,Z 735.949,A -85,B 0,C 180,E1 15084.52,E2 15084.52} C_VEL
LIN {X 0,Y 396.609,Z 759.003,A -85,B 0,C 180,E1 15083.863,E2 15083.863} C_VEL
LIN {X 0,Y 392.799,Z 781.704,A -85,B 0,C 180,E1 15083.004,E2 15083.004} C_VEL
LIN {X 0,Y 388.754,Z 801.57,A -85,B 0,C 180,E1 15082.031,E2 15082.031} C_VEL
LIN {X 0,Y 383.698,Z 823.32,A -85,B 0,C 180,E1 15080.712,E2 15080.712} C_VEL
LIN {X 0,Y 378.611,Z 842.492,A -85,B 0,C 180,E1 15079.286,E2 15079.286} C_VEL
LIN {X 0,Y 372.7,Z 862.973,A -85,B 0,C 180,E1 15077.465,E2 15077.465} C_VEL
LIN {X 0,Y 366.827,Z 881.672,A -85,B 0,C 180,E1 15075.464,E2 15075.464} C_VEL
LIN {X 0,Y 360.295,Z 901.398,A -85,B 0,C 180,E1 15072.948,E2 15072.948} C_VEL
LIN {X 0,Y 354.268,Z 919.091,A -85,B 0,C 180,E1 15070.268,E2 15070.268} C_VEL
LIN {X 0,Y 348.715,Z 934.851,A -85,B 0,C 180,E1 15067.418,E2 15067.418} C_VEL
LIN {X 0,Y 343.486,Z 950.137,A -85,B 0,C 180,E1 15064.185,E2 15064.185} C_VEL
LIN {X 0,Y 339.089,Z 963.293,A -85,B 0,C 180,E1 15060.872,E2 15060.872} C_VEL
LIN {X 0,Y 335.067,Z 976.309,A -85,B 0,C 180,E1 15056.977,E2 15056.977} C_VEL
LIN {X 0,Y 332.222,Z 986.787,A -85,B 0,C 180,E1 15053.224,E2 15053.224} C_VEL
LIN {X 0,Y 330.237,Z 995.339,A -85,B 0,C 180,E1 15049.458,E2 15049.458} C_VEL
LIN {X 0,Y 328.972,Z 1002.374,A -85,B 0,C 180,E1 15045.698,E2 15045.698} C_VEL
LIN {X 0,Y 328.279,Z 1007.72,A -85,B 0,C 180,E1 15041.957,E2 15041.957} C_VEL
LIN {X 0,Y 328.03,Z 1011.512,A -85,B 0,C 180,E1 15038.417,E2 15038.417} C_VEL
LIN {X 0,Y 327.943,Z 1014.143,A -85,B 0,C 180,E1 15034.551,E2 15034.551} C_VEL
LIN {X 0,Y 327.949,Z 1015.149,A -85,B 0,C 180,E1 15031.227,E2 15031.227} C_VEL
LIN {X 0,Y 327.953,Z 1015.057,A -85,B 0,C 180,E1 15027.908,E2 15027.908} C_VEL
LIN {X 0,Y 327.95,Z 1013.454,A -85,B 0,C 180,E1 15024.055,E2 15024.055} C_VEL
LIN {X 0,Y 328.06,Z 1010.82,A -85,B 0,C 180,E1 15020.709,E2 15020.709} C_VEL
LIN {X 0,Y 328.47,Z 1006.352,A -85,B 0,C 180,E1 15016.808,E2 15016.808} C_VEL
LIN {X 0,Y 329.334,Z 1000.437,A -85,B 0,C 180,E1 15013.06,E2 15013.06} C_VEL
